# B&R Automation Studio project AutomatedPongGame (part 2)

#### basic.c
```c
/*******************************************************************
 * COPYRIGHT -- Bernecker + Rainer
 ********************************************************************
 * PROGRAM: Basic
 * File: Basic.c
 * Author: Bernecker + Rainer
 * Created: December 01, 2009
 ********************************************************************
 * Implementation of Program Basic
 ********************************************************************/

#ifdef _DEFAULT_INCLUDES
 #include <AsDefault.h>
#endif
#include <string.h>

/* defines of the state-constants */
#define STATE_WAIT              0
#define STATE_POWER_ON          1
#define STATE_HOME              2

#define STATE_READY             10
#define STATE_HALT              11
#define STATE_STOP              12
#define STATE_JOG_POSITIVE      13
#define STATE_JOG_NEGATIVE      14
#define STATE_MOVE_ABSOLUTE     15
#define STATE_MOVE_ADDITIVE     16
#define STATE_MOVE_VELOCITY     17

#define STATE_ERROR_AXIS        100
#define STATE_ERROR             101
#define STATE_ERROR_RESET       102

_INIT void BasicControl_init(void)
{

/* get axis object */
Axis1Obj = (UDINT)&gAxis01;

AxisStep = STATE_WAIT;  /* start step */

BasicControl.Parameter.Velocity              = 1000;  /*velocity for movement*/
BasicControl.Parameter.Acceleration          = 5000;  /*acceleration for movement*/
BasicControl.Parameter.Deceleration          = 5000;  /*deceleration for movement*/
BasicControl.Parameter.JogVelocity           = 400;   /*velocity for jogging */

}

_CYCLIC void BasicControl_cyclic(void)
{

/***************************************************************
        Control Sequence
***************************************************************/

/* status information is read before the step sequencer to attain a shorter reaction time */
/************************ MC_READSTATUS *************************/
MC_ReadStatus_0.Enable = !MC_ReadStatus_0.Error;
MC_ReadStatus_0.Axis = Axis1Obj;
MC_ReadStatus(&MC_ReadStatus_0);
BasicControl.AxisState.Disabled             = MC_ReadStatus_0.Disabled;
BasicControl.AxisState.StandStill           = MC_ReadStatus_0.StandStill;
BasicControl.AxisState.Stopping             = MC_ReadStatus_0.Stopping;
BasicControl.AxisState.Homing               = MC_ReadStatus_0.Homing;
BasicControl.AxisState.DiscreteMotion       = MC_ReadStatus_0.DiscreteMotion;
BasicControl.AxisState.ContinuousMotion     = MC_ReadStatus_0.ContinuousMotion;
BasicControl.AxisState.SynchronizedMotion   = MC_ReadStatus_0.SynchronizedMotion;
BasicControl.AxisState.ErrorStop            = MC_ReadStatus_0.Errorstop;

/********************MC_BR_READDRIVESTATUS***********************/
MC_BR_ReadDriveStatus_0.Enable = !MC_BR_ReadDriveStatus_0.Error;
MC_BR_ReadDriveStatus_0.Axis = Axis1Obj;
MC_BR_ReadDriveStatus_0.AdrDriveStatus = (UDINT)&(BasicControl.Status.DriveStatus);
MC_BR_ReadDriveStatus(&MC_BR_ReadDriveStatus_0);

/******************** MC_READACTUALPOSITION *********************/
MC_ReadActualPosition_0.Enable = (!MC_ReadActualPosition_0.Error);
MC_ReadActualPosition_0.Axis = Axis1Obj;
MC_ReadActualPosition(&MC_ReadActualPosition_0);
if(MC_ReadActualPosition_0.Valid == 1)
{
    BasicControl.Status.ActPosition = MC_ReadActualPosition_0.Position;
}

/******************** MC_READACTUALVELOCITY *********************/
MC_ReadActualVelocity_0.Enable = (!MC_ReadActualVelocity_0.Error);
MC_ReadActualVelocity_0.Axis = Axis1Obj;
MC_ReadActualVelocity(&MC_ReadActualVelocity_0);
if(MC_ReadActualVelocity_0.Valid == 1)
{
    BasicControl.Status.ActVelocity = MC_ReadActualVelocity_0.Velocity;
}

/************************ MC_READAXISERROR **********************/
MC_ReadAxisError_0.Enable = !MC_ReadAxisError_0.Error;
MC_ReadAxisError_0.Axis = Axis1Obj;
MC_ReadAxisError_0.DataAddress = (UDINT)&(BasicControl.Status.ErrorText);
MC_ReadAxisError_0.DataLength = sizeof(BasicControl.Status.ErrorText);
strcpy((void*)&MC_ReadAxisError_0.DataObjectName,"acp10etxen");
MC_ReadAxisError(&MC_ReadAxisError_0);

/**************** CHECK FOR GENERAL AXIS ERROR ******************/
    if ((MC_ReadAxisError_0.AxisErrorID != 0) && (MC_ReadAxisError_0.Valid == 1))
    {
        AxisStep = STATE_ERROR_AXIS;
    }
/***************** CHECK IF POWER SHOULD BE OFF *******************/
    else if ((BasicControl.Command.Power == 0) && (MC_ReadAxisError_0.Valid == 1))
    {
        if ((MC_ReadStatus_0.Errorstop == 1) && (MC_ReadStatus_0.Valid == 1))
        {
            AxisStep = STATE_ERROR_RESET;
        }
        else
        {
            AxisStep = STATE_WAIT;
        }
    }

/* central monitoring of stop command attains a shorter reaction time in case of emergency stop */
/******************CHECK for STOP COMMAND************************/
    if (BasicControl.Command.Stop == 1)
    {
        if ((AxisStep >= STATE_HOME) && (AxisStep <= STATE_ERROR))
        {
            /* reset all FB execute inputs we use */
            MC_Home_0.Execute = 0;
            MC_Stop_0.Execute = 0;
            MC_MoveAbsolute_0.Execute = 0;
            MC_MoveAdditive_0.Execute = 0;
            MC_MoveVelocity_0.Execute = 0;
            MC_Halt_0.Execute = 0;
            MC_ReadAxisError_0.Acknowledge = 0;
            MC_Reset_0.Execute = 0;

            /* reset user commands */
            BasicControl.Command.Halt = 0;
            BasicControl.Command.Home = 0;
            BasicControl.Command.MoveJogPos = 0;
            BasicControl.Command.MoveJogNeg = 0;
            BasicControl.Command.MoveVelocity = 0;
            BasicControl.Command.MoveAbsolute = 0;
            BasicControl.Command.MoveAdditive = 0;
            AxisStep = STATE_STOP;
        }
    }

switch(AxisStep)
{
/******************** WAIT *************************/
    case STATE_WAIT:  /* STATE: Wait */
        if (BasicControl.Command.Power == 1)
        {
            AxisStep = STATE_POWER_ON;
        }
        else
        {
            MC_Power_0.Enable = 0;
        }

        /* reset all FB execute inputs we use */
        MC_Home_0.Execute = 0;
        MC_Stop_0.Execute = 0;
        MC_MoveAbsolute_0.Execute = 0;
        MC_MoveAdditive_0.Execute = 0;
        MC_MoveVelocity_0.Execute = 0;
        MC_Halt_0.Execute = 0;
        MC_ReadAxisError_0.Acknowledge = 0;
        MC_Reset_0.Execute = 0;

        /* reset user commands */
        BasicControl.Command.Halt = 0;
        BasicControl.Command.Home = 0;
        BasicControl.Command.MoveJogPos = 0;
        BasicControl.Command.MoveJogNeg = 0;
        BasicControl.Command.MoveVelocity = 0;
        BasicControl.Command.MoveAbsolute = 0;
        BasicControl.Command.MoveAdditive = 0;

        BasicControl.Status.ErrorID = 0;
    break;

/******************** POWER ON **********************/
    case STATE_POWER_ON:  /* STATE: Power on */
        MC_Power_0.Enable = 1;
        if (MC_Power_0.Status == 1)
        {
            AxisStep = STATE_READY;
        }
        /* if a power error occured go to error state */
        if (MC_Power_0.Error == 1)
        {
            BasicControl.Status.ErrorID = MC_Power_0.ErrorID;
            AxisStep = STATE_ERROR;
        }
    break;

/******************** READY **********************/
    case STATE_READY:  /* STATE: Waiting for commands */
        if (BasicControl.Command.Home == 1)
        {
            BasicControl.Command.Home = 0;
            AxisStep = STATE_HOME;
        }
        else if (BasicControl.Command.Stop == 1)
        {
            AxisStep = STATE_STOP;
        }
        else if (BasicControl.Command.MoveJogPos == 1)
        {
            AxisStep = STATE_JOG_POSITIVE;
        }
        else if (BasicControl.Command.MoveJogNeg == 1)
        {
            AxisStep = STATE_JOG_NEGATIVE;
        }
        else if (BasicControl.Command.MoveAbsolute == 1)
        {
            BasicControl.Command.MoveAbsolute = 0;
            AxisStep = STATE_MOVE_ABSOLUTE;
        }
        else if (BasicControl.Command.MoveAdditive == 1)
        {
            BasicControl.Command.MoveAdditive = 0;
            AxisStep = STATE_MOVE_ADDITIVE;
        }
        else if (BasicControl.Command.MoveVelocity == 1)
        {
            BasicControl.Command.MoveVelocity = 0;
            AxisStep = STATE_MOVE_VELOCITY;
        }
        else if (BasicControl.Command.Halt == 1)
        {
            BasicControl.Command.Halt = 0;
            AxisStep = STATE_HALT;
        }
    break;

/******************** HOME **********************/
    case STATE_HOME:  /* STATE: start homing process */
        MC_Home_0.Position = BasicControl.Parameter.HomePosition;
        MC_Home_0.HomingMode = BasicControl.Parameter.HomeMode;
        MC_Home_0.Execute = 1;
        if (MC_Home_0.Done == 1)
        {
            MC_Home_0.Execute = 0;
            AxisStep = STATE_READY;
        }
        /* if a homing error occured go to error state */
        if (MC_Home_0.Error == 1)
        {
            MC_Home_0.Execute = 0;
            BasicControl.Status.ErrorID = MC_Home_0.ErrorID;
            AxisStep = STATE_ERROR;
        }
    break;

/************************HALT MOVEMENT**************************/
    case STATE_HALT:  /* STATE: Stop the active movement */
        MC_Halt_0.Deceleration = BasicControl.Parameter.Deceleration;
        MC_Halt_0.Execute = 1;
        if (MC_Halt_0.Done == 1)
        {
            MC_Halt_0.Execute = 0;
            AxisStep = STATE_READY;
        }
        /*check if error occured */
        if (MC_Halt_0.Error == 1)
        {
            MC_Halt_0.Execute = 0;
            BasicControl.Status.ErrorID = MC_Halt_0.ErrorID;
            AxisStep = STATE_ERROR;
        }
    break;

/*********************** STOP MOVEMENT *************************/
    case STATE_STOP: /* STATE: Stop movement as long as command is set */
        MC_Stop_0.Deceleration = BasicControl.Parameter.Deceleration;
        MC_Stop_0.Execute = 1;
        /* if axis is stopped go to ready state */
        if ((MC_Stop_0.Done == 1) && (BasicControl.Command.Stop == 0))
        {
            MC_Stop_0.Execute = 0;
            AxisStep = STATE_READY;
        }
        /* check if error occured */
        if (MC_Stop_0.Error == 1)
        {
            BasicControl.Status.ErrorID = MC_Stop_0.ErrorID;
            MC_Stop_0.Execute = 0;
            AxisStep = STATE_ERROR;
        }
    break;

/******************** START JOG MOVEMENT POSITVE **********************/
    case STATE_JOG_POSITIVE:  /* STATE: Start jog movement in positive direction */
        MC_MoveVelocity_0.Velocity      = BasicControl.Parameter.JogVelocity;
        MC_MoveVelocity_0.Acceleration  = BasicControl.Parameter.Acceleration;
        MC_MoveVelocity_0.Deceleration  = BasicControl.Parameter.Deceleration;
        MC_MoveVelocity_0.Direction     = mcPOSITIVE_DIR;
        MC_MoveVelocity_0.Execute = 1;
        /* check if jog movement should be stopped */
        if (BasicControl.Command.MoveJogPos == 0)
        {
            MC_MoveVelocity_0.Execute = 0;
            AxisStep = STATE_HALT;
        }
        /* check if error occured */
        if (MC_MoveVelocity_0.Error == 1)
        {
            BasicControl.Status.ErrorID = MC_MoveVelocity_0.ErrorID;
            MC_MoveVelocity_0.Execute = 0;
            AxisStep = STATE_ERROR;
        }
    break;

/******************** START JOG MOVEMENT NEGATIVE **********************/
    case STATE_JOG_NEGATIVE:  /* STATE: Start jog movement in negative direction */
        MC_MoveVelocity_0.Velocity      = BasicControl.Parameter.JogVelocity;
        MC_MoveVelocity_0.Acceleration  = BasicControl.Parameter.Acceleration;
        MC_MoveVelocity_0.Deceleration  = BasicControl.Parameter.Deceleration;
        MC_MoveVelocity_0.Direction     = mcNEGATIVE_DIR;
        MC_MoveVelocity_0.Execute = 1;
        /* check if jog movement should be stopped */
        if (BasicControl.Command.MoveJogNeg == 0)
        {
            MC_MoveVelocity_0.Execute = 0;
            AxisStep = STATE_HALT;
        }
        /* check if error occured */
        if (MC_MoveVelocity_0.Error == 1)
        {
            BasicControl.Status.ErrorID = MC_MoveVelocity_0.ErrorID;
            MC_MoveVelocity_0.Execute = 0;
            AxisStep = STATE_ERROR;
        }
    break;

/******************** START ABSOLUTE MOVEMENT **********************/
    case STATE_MOVE_ABSOLUTE:  /* STATE: Start absolute movement */
        MC_MoveAbsolute_0.Position      = BasicControl.Parameter.Position;
        MC_MoveAbsolute_0.Velocity      = BasicControl.Parameter.Velocity;
        MC_MoveAbsolute_0.Acceleration  = BasicControl.Parameter.Acceleration;
        MC_MoveAbsolute_0.Deceleration  = BasicControl.Parameter.Deceleration;
        MC_MoveAbsolute_0.Direction     = BasicControl.Parameter.Direction;
        MC_MoveAbsolute_0.Execute = 1;
        /* check if commanded position is reached */
        if (BasicControl.Command.Halt == 1)
        {
            BasicControl.Command.Halt = 0;
            MC_MoveAbsolute_0.Execute = 0;
            AxisStep = STATE_HALT;
        }
        else if (MC_MoveAbsolute_0.Done == 1)
        {
            MC_MoveAbsolute_0.Execute = 0;
             AxisStep = STATE_READY;
        }
        /* check if error occured */
        if (MC_MoveAbsolute_0.Error == 1)
        {
            BasicControl.Status.ErrorID = MC_MoveAbsolute_0.ErrorID;
            MC_MoveAbsolute_0.Execute = 0;
            AxisStep = STATE_ERROR;
        }
    break;

/******************** START ADDITIVE MOVEMENT **********************/
    case STATE_MOVE_ADDITIVE:  /* STATE: Start additive movement */
        MC_MoveAdditive_0.Distance      = BasicControl.Parameter.Distance;
        MC_MoveAdditive_0.Velocity      = BasicControl.Parameter.Velocity;
        MC_MoveAdditive_0.Acceleration  = BasicControl.Parameter.Acceleration;
        MC_MoveAdditive_0.Deceleration  = BasicControl.Parameter.Deceleration;
        MC_MoveAdditive_0.Execute = 1;
        /* check if commanded distance is reached */
        if (BasicControl.Command.Halt == 1)
        {
            BasicControl.Command.Halt = 0;
            MC_MoveAdditive_0.Execute = 0;
            AxisStep = STATE_HALT;
        }
        else if (MC_MoveAdditive_0.Done == 1)
        {
            MC_MoveAdditive_0.Execute = 0;
             AxisStep = STATE_READY;
        }
        /* check if error occured */
        if (MC_MoveAdditive_0.Error == 1)
        {
            BasicControl.Status.ErrorID = MC_MoveAdditive_0.ErrorID;
            MC_MoveAdditive_0.Execute = 0;
            AxisStep = STATE_ERROR;
        }
    break;

/******************** START VELOCITY MOVEMENT **********************/
    case STATE_MOVE_VELOCITY:  /* STATE: Start velocity movement */
        MC_MoveVelocity_0.Velocity      = BasicControl.Parameter.Velocity;
        MC_MoveVelocity_0.Acceleration  = BasicControl.Parameter.Acceleration;
        MC_MoveVelocity_0.Deceleration  = BasicControl.Parameter.Deceleration;
        MC_MoveVelocity_0.Direction     = BasicControl.Parameter.Direction;
        MC_MoveVelocity_0.Execute = 1;
        /* check if commanded velocity is reached */
        if (BasicControl.Command.Halt == 1)
        {
            BasicControl.Command.Halt = 0;
            MC_MoveVelocity_0.Execute = 0;
            AxisStep = STATE_HALT;
        }
        else if (MC_MoveVelocity_0.InVelocity == 1)
        {
            MC_MoveVelocity_0.Execute = 0;
             AxisStep = STATE_READY;
        }
        /* check if error occured */
        if (MC_MoveVelocity_0.Error == 1)
        {
            BasicControl.Status.ErrorID = MC_MoveVelocity_0.ErrorID;
            MC_MoveVelocity_0.Execute = 0;
            AxisStep = STATE_ERROR;
        }
    break;

/******************** FB-ERROR OCCURED *************************/
    case STATE_ERROR:  /* STATE: Error */
        /* check if FB indicates an axis error */
        if (MC_ReadAxisError_0.AxisErrorCount != 0)
        {
            AxisStep = STATE_ERROR_AXIS;
        }
        else
        {
            if (BasicControl.Command.ErrorAcknowledge == 1)
            {
                BasicControl.Command.ErrorAcknowledge = 0;
                BasicControl.Status.ErrorID = 0;
                /* reset axis if it is in axis state ErrorStop */
                if ((MC_ReadStatus_0.Errorstop == 1) && (MC_ReadStatus_0.Valid == 1))
                {
                    AxisStep = STATE_ERROR_RESET;
                }
                else
                {
                    AxisStep = STATE_WAIT;
                }
            }
        }
    break;

/******************** AXIS-ERROR OCCURED *************************/
    case STATE_ERROR_AXIS:  /* STATE: Axis Error */
        if (MC_ReadAxisError_0.Valid == 1)
        {
            if (MC_ReadAxisError_0.AxisErrorID != 0)
            {
                BasicControl.Status.ErrorID = MC_ReadAxisError_0.AxisErrorID;
            }
            MC_ReadAxisError_0.Acknowledge = 0;
            if (BasicControl.Command.ErrorAcknowledge == 1)
            {
                BasicControl.Command.ErrorAcknowledge = 0;
                /* acknowledge axis error */
                if (MC_ReadAxisError_0.AxisErrorID != 0)
                {
                    MC_ReadAxisError_0.Acknowledge = 1;
                }
            }
            if (MC_ReadAxisError_0.AxisErrorCount == 0)
            {
                BasicControl.Status.ErrorID = 0;
                /* reset axis if it is in axis state ErrorStop */
                if ((MC_ReadStatus_0.Errorstop == 1) && (MC_ReadStatus_0.Valid == 1))
                {
                    AxisStep = STATE_ERROR_RESET;
                }
                else
                {
                    AxisStep = STATE_WAIT;
                }
            }
        }
    break;

/******************** RESET DONE *************************/
    case STATE_ERROR_RESET:  /* STATE: Wait for reset done */
        MC_Reset_0.Execute = 1;
        /* reset MC_Power.Enable if this FB is in Error*/
        if(MC_Power_0.Error == 1)
        {
            MC_Power_0.Enable = 0;
        }
        if(MC_Reset_0.Done == 1)
        {
            MC_Reset_0.Execute = 0;
            AxisStep = STATE_WAIT;
        }
        else if (MC_Reset_0.Error == 1)
        {
            MC_Reset_0.Execute = 0;
            AxisStep = STATE_ERROR;
        }
    break;

/******************** SEQUENCE END *************************/
}

/***************************************************************
        Function Block Calls
***************************************************************/

/************************** MC_POWER ****************************/
MC_Power_0.Axis = Axis1Obj;  /* pointer to axis */
MC_Power(&MC_Power_0);

/************************** MC_HOME *****************************/
MC_Home_0.Axis = Axis1Obj;
MC_Home(&MC_Home_0);

/********************** MC_MOVEABSOLUTE *************************/
MC_MoveAbsolute_0.Axis = Axis1Obj;
MC_MoveAbsolute(&MC_MoveAbsolute_0);

/********************** MC_MOVEADDITIVE *************************/
MC_MoveAdditive_0.Axis = Axis1Obj;
MC_MoveAdditive(&MC_MoveAdditive_0);

/********************** MC_MOVEVELOCITY *************************/
MC_MoveVelocity_0.Axis = Axis1Obj;
MC_MoveVelocity(&MC_MoveVelocity_0);

/************************** MC_STOP *****************************/
MC_Stop_0.Axis = Axis1Obj;
MC_Stop(&MC_Stop_0);

/**************************MC_HALT*******************************/
MC_Halt_0.Axis = Axis1Obj;
MC_Halt(&MC_Halt_0);

/************************** MC_RESET ****************************/
MC_Reset_0.Axis = Axis1Obj;
MC_Reset(&MC_Reset_0);

}
```

#### Cyclic.cpp
```cpp
#ifdef _DEFAULT_INCLUDES
	#include <AsDefault.h>
#endif
#include <string.h>

/* defines of the state-constants */
#define STATE_WAIT              0
#define STATE_POWER_ON          1
#define STATE_HOME              2

#define STATE_READY             10
#define STATE_HALT              11
#define STATE_STOP              12
#define STATE_JOG_POSITIVE      13
#define STATE_JOG_NEGATIVE      14
#define STATE_MOVE_ABSOLUTE     15
#define STATE_MOVE_ADDITIVE     16
#define STATE_MOVE_VELOCITY     17

#define STATE_ERROR_AXIS        100
#define STATE_ERROR             101
#define STATE_ERROR_RESET       102

#define RED_COLOR 51
#define GREEN_COLOR 10

#define MIDDELPUNT_TRAPPER_OFFSET 15
//#define ACTPOSITION_TO_MM 0.0784

unsigned long bur_heap_size = 0xFFFF;

void _CYCLIC ProgramCyclic(void)
{
	/***************************************************************
        Control Sequence
	***************************************************************/

	/* status information is read before the step sequencer to attain a shorter reaction time */
	/************************ MC_READSTATUS *************************/
	MC_ReadStatus_0.Enable = !MC_ReadStatus_0.Error;
	MC_ReadStatus_0.Axis = Axis1Obj;
	MC_ReadStatus(&MC_ReadStatus_0);
	BasicControl.AxisState.Disabled             = MC_ReadStatus_0.Disabled;
	BasicControl.AxisState.StandStill           = MC_ReadStatus_0.StandStill;
	BasicControl.AxisState.Stopping             = MC_ReadStatus_0.Stopping;
	BasicControl.AxisState.Homing               = MC_ReadStatus_0.Homing;
	BasicControl.AxisState.DiscreteMotion       = MC_ReadStatus_0.DiscreteMotion;
	BasicControl.AxisState.ContinuousMotion     = MC_ReadStatus_0.ContinuousMotion;
	BasicControl.AxisState.SynchronizedMotion   = MC_ReadStatus_0.SynchronizedMotion;
	BasicControl.AxisState.ErrorStop            = MC_ReadStatus_0.Errorstop;

	/********************MC_BR_READDRIVESTATUS***********************/
	MC_BR_ReadDriveStatus_0.Enable = !MC_BR_ReadDriveStatus_0.Error;
	MC_BR_ReadDriveStatus_0.Axis = Axis1Obj;
	MC_BR_ReadDriveStatus_0.AdrDriveStatus = (UDINT)&(BasicControl.Status.DriveStatus);
	MC_BR_ReadDriveStatus(&MC_BR_ReadDriveStatus_0);

	/******************** MC_READACTUALPOSITION *********************/
	MC_ReadActualPosition_0.Enable = (!MC_ReadActualPosition_0.Error);
	MC_ReadActualPosition_0.Axis = Axis1Obj;
	MC_ReadActualPosition(&MC_ReadActualPosition_0);
	if(MC_ReadActualPosition_0.Valid == 1)
	{
		BasicControl.Status.ActPosition = MC_ReadActualPosition_0.Position;
	}

	/******************** MC_READACTUALVELOCITY *********************/
	MC_ReadActualVelocity_0.Enable = (!MC_ReadActualVelocity_0.Error);
	MC_ReadActualVelocity_0.Axis = Axis1Obj;
	MC_ReadActualVelocity(&MC_ReadActualVelocity_0);
	if(MC_ReadActualVelocity_0.Valid == 1)
	{
		BasicControl.Status.ActVelocity = MC_ReadActualVelocity_0.Velocity;
	}

	/************************ MC_READAXISERROR **********************/
	MC_ReadAxisError_0.Enable = !MC_ReadAxisError_0.Error;
	MC_ReadAxisError_0.Axis = Axis1Obj;
	MC_ReadAxisError_0.DataAddress = (UDINT)&(BasicControl.Status.ErrorText);
	MC_ReadAxisError_0.DataLength = sizeof(BasicControl.Status.ErrorText);
	strcpy(MC_ReadAxisError_0.DataObjectName,"acp10etxen");
	MC_ReadAxisError(&MC_ReadAxisError_0);

	/**************** CHECK FOR GENERAL AXIS ERROR ******************/
	if ((MC_ReadAxisError_0.AxisErrorID != 0) && (MC_ReadAxisError_0.Valid == 1))
	{
		AxisStep = STATE_ERROR_AXIS;
	}
		/***************** CHECK IF POWER SHOULD BE OFF *******************/
	else if ((BasicControl.Command.Power == 0) && (MC_ReadAxisError_0.Valid == 1))
	{
		if ((MC_ReadStatus_0.Errorstop == 1) && (MC_ReadStatus_0.Valid == 1))
		{
			AxisStep = STATE_ERROR_RESET;
		}
		else
		{
			AxisStep = STATE_WAIT;
		}
	}

	/* central monitoring of stop command attains a shorter reaction time in case of emergency stop */
	/******************CHECK for STOP COMMAND************************/
	if (BasicControl.Command.Stop == 1)
	{
		if ((AxisStep >= STATE_HOME) && (AxisStep <= STATE_ERROR))
		{
			/* reset all FB execute inputs we use */
			MC_Home_0.Execute = 0;
			MC_Stop_0.Execute = 0;
			MC_MoveAbsolute_0.Execute = 0;
			MC_MoveAdditive_0.Execute = 0;
			MC_MoveVelocity_0.Execute = 0;
			MC_Halt_0.Execute = 0;
			MC_ReadAxisError_0.Acknowledge = 0;
			MC_Reset_0.Execute = 0;

			/* reset user commands */
			BasicControl.Command.Halt = 0;
			BasicControl.Command.Home = 0;
			BasicControl.Command.MoveJogPos = 0;
			BasicControl.Command.MoveJogNeg = 0;
			BasicControl.Command.MoveVelocity = 0;
			BasicControl.Command.MoveAbsolute = 0;
			BasicControl.Command.MoveAdditive = 0;
			AxisStep = STATE_STOP;
		}
	}

	switch(AxisStep)
	{
		/******************** WAIT *************************/
		case STATE_WAIT:  /* STATE: Wait */
			if (BasicControl.Command.Power == 1)
			{
				AxisStep = STATE_POWER_ON;
			}
			else
			{
				MC_Power_0.Enable = 0;
			}

			/* reset all FB execute inputs we use */
			MC_Home_0.Execute = 0;
			MC_Stop_0.Execute = 0;
			MC_MoveAbsolute_0.Execute = 0;
			MC_MoveAdditive_0.Execute = 0;
			MC_MoveVelocity_0.Execute = 0;
			MC_Halt_0.Execute = 0;
			MC_ReadAxisError_0.Acknowledge = 0;
			MC_Reset_0.Execute = 0;

			/* reset user commands */
			BasicControl.Command.Halt = 0;
			BasicControl.Command.Home = 0;
			BasicControl.Command.MoveJogPos = 0;
			BasicControl.Command.MoveJogNeg = 0;
			BasicControl.Command.MoveVelocity = 0;
			BasicControl.Command.MoveAbsolute = 0;
			BasicControl.Command.MoveAdditive = 0;

			BasicControl.Status.ErrorID = 0;
			break;

		/******************** POWER ON **********************/
		case STATE_POWER_ON:  /* STATE: Power on */
			MC_Power_0.Enable = 1;
			if (MC_Power_0.Status == 1)
			{
				AxisStep = STATE_READY;
			}
			/* if a power error occured go to error state */
			if (MC_Power_0.Error == 1)
			{
				BasicControl.Status.ErrorID = MC_Power_0.ErrorID;
				AxisStep = STATE_ERROR;
			}
			break;

		/******************** READY **********************/
		case STATE_READY:  /* STATE: Waiting for commands */
			if (BasicControl.Command.Home == 1)
			{
				BasicControl.Command.Home = 0;
				AxisStep = STATE_HOME;
			}
			else if (BasicControl.Command.Stop == 1)
			{
				AxisStep = STATE_STOP;
			}
			else if (BasicControl.Command.MoveJogPos == 1)
			{
				AxisStep = STATE_JOG_POSITIVE;
			}
			else if (BasicControl.Command.MoveJogNeg == 1)
			{
				AxisStep = STATE_JOG_NEGATIVE;
			}
			else if (BasicControl.Command.MoveAbsolute == 1)
			{
				BasicControl.Command.MoveAbsolute = 0;
				AxisStep = STATE_MOVE_ABSOLUTE;
			}
			else if (BasicControl.Command.MoveAdditive == 1)
			{
				BasicControl.Command.MoveAdditive = 0;
				AxisStep = STATE_MOVE_ADDITIVE;
			}
			else if (BasicControl.Command.MoveVelocity == 1)
			{
				BasicControl.Command.MoveVelocity = 0;
				AxisStep = STATE_MOVE_VELOCITY;
			}
			else if (BasicControl.Command.Halt == 1)
			{
				BasicControl.Command.Halt = 0;
				AxisStep = STATE_HALT;
			}
			break;

		/******************** HOME **********************/
		case STATE_HOME:  /* STATE: start homing process */
			MC_Home_0.Position = BasicControl.Parameter.HomePosition;
			MC_Home_0.HomingMode = BasicControl.Parameter.HomeMode;
			MC_Home_0.Execute = 1;
			if (MC_Home_0.Done == 1)
			{
				MC_Home_0.Execute = 0;
				AxisStep = STATE_READY;
			}
			/* if a homing error occured go to error state */
			if (MC_Home_0.Error == 1)
			{
				MC_Home_0.Execute = 0;
				BasicControl.Status.ErrorID = MC_Home_0.ErrorID;
				AxisStep = STATE_ERROR;
			}
			break;

		/************************HALT MOVEMENT**************************/
		case STATE_HALT:  /* STATE: Stop the active movement */
			MC_Halt_0.Deceleration = BasicControl.Parameter.Deceleration;
			MC_Halt_0.Execute = 1;
			if (MC_Halt_0.Done == 1)
			{
				MC_Halt_0.Execute = 0;
				AxisStep = STATE_READY;
			}
			/*check if error occured */
			if (MC_Halt_0.Error == 1)
			{
				MC_Halt_0.Execute = 0;
				BasicControl.Status.ErrorID = MC_Halt_0.ErrorID;
				AxisStep = STATE_ERROR;
			}
			break;

		/*********************** STOP MOVEMENT *************************/
		case STATE_STOP: /* STATE: Stop movement as long as command is set */
			MC_Stop_0.Deceleration = BasicControl.Parameter.Deceleration;
			MC_Stop_0.Execute = 1;
			/* if axis is stopped go to ready state */
			if ((MC_Stop_0.Done == 1) && (BasicControl.Command.Stop == 0))
			{
				MC_Stop_0.Execute = 0;
				AxisStep = STATE_READY;
			}
			/* check if error occured */
			if (MC_Stop_0.Error == 1)
			{
				BasicControl.Status.ErrorID = MC_Stop_0.ErrorID;
				MC_Stop_0.Execute = 0;
				AxisStep = STATE_ERROR;
			}
			break;

		/******************** START JOG MOVEMENT POSITVE **********************/
		case STATE_JOG_POSITIVE:  /* STATE: Start jog movement in positive direction */
			MC_MoveVelocity_0.Velocity      = BasicControl.Parameter.JogVelocity;
			MC_MoveVelocity_0.Acceleration  = BasicControl.Parameter.Acceleration;
			MC_MoveVelocity_0.Deceleration  = BasicControl.Parameter.Deceleration;
			MC_MoveVelocity_0.Direction     = mcPOSITIVE_DIR;
			MC_MoveVelocity_0.Execute = 1;
			/* check if jog movement should be stopped */
			if (BasicControl.Command.MoveJogPos == 0)
			{
				MC_MoveVelocity_0.Execute = 0;
				AxisStep = STATE_HALT;
			}
			/* check if error occured */
			if (MC_MoveVelocity_0.Error == 1)
			{
				BasicControl.Status.ErrorID = MC_MoveVelocity_0.ErrorID;
				MC_MoveVelocity_0.Execute = 0;
				AxisStep = STATE_ERROR;
			}
			break;

		/******************** START JOG MOVEMENT NEGATIVE **********************/
		case STATE_JOG_NEGATIVE:  /* STATE: Start jog movement in negative direction */
			MC_MoveVelocity_0.Velocity      = BasicControl.Parameter.JogVelocity;
			MC_MoveVelocity_0.Acceleration  = BasicControl.Parameter.Acceleration;
			MC_MoveVelocity_0.Deceleration  = BasicControl.Parameter.Deceleration;
			MC_MoveVelocity_0.Direction     = mcNEGATIVE_DIR;
			MC_MoveVelocity_0.Execute = 1;
			/* check if jog movement should be stopped */
			if (BasicControl.Command.MoveJogNeg == 0)
			{
				MC_MoveVelocity_0.Execute = 0;
				AxisStep = STATE_HALT;
			}
			/* check if error occured */
			if (MC_MoveVelocity_0.Error == 1)
			{
				BasicControl.Status.ErrorID = MC_MoveVelocity_0.ErrorID;
				MC_MoveVelocity_0.Execute = 0;
				AxisStep = STATE_ERROR;
			}
			break;

		/******************** START ABSOLUTE MOVEMENT **********************/
		case STATE_MOVE_ABSOLUTE:  /* STATE: Start absolute movement */
			MC_MoveAbsolute_0.Position      = BasicControl.Parameter.Position;
			MC_MoveAbsolute_0.Velocity      = BasicControl.Parameter.Velocity;
			MC_MoveAbsolute_0.Acceleration  = BasicControl.Parameter.Acceleration;
			MC_MoveAbsolute_0.Deceleration  = BasicControl.Parameter.Deceleration;
			MC_MoveAbsolute_0.Direction     = BasicControl.Parameter.Direction;
			MC_MoveAbsolute_0.Execute = 1;
			/* check if commanded position is reached */
			if (BasicControl.Command.Halt == 1)
			{
				BasicControl.Command.Halt = 0;
				MC_MoveAbsolute_0.Execute = 0;
				AxisStep = STATE_HALT;
			}
			else if (MC_MoveAbsolute_0.Done == 1)
			{
				MC_MoveAbsolute_0.Execute = 0;
				AxisStep = STATE_READY;
			}
			/* check if error occured */
			if (MC_MoveAbsolute_0.Error == 1)
			{
				BasicControl.Status.ErrorID = MC_MoveAbsolute_0.ErrorID;
				MC_MoveAbsolute_0.Execute = 0;
				AxisStep = STATE_ERROR;
			}
			break;

		/******************** START ADDITIVE MOVEMENT **********************/
		case STATE_MOVE_ADDITIVE:  /* STATE: Start additive movement */
			MC_MoveAdditive_0.Distance      = BasicControl.Parameter.Distance;
			MC_MoveAdditive_0.Velocity      = BasicControl.Parameter.Velocity;
			MC_MoveAdditive_0.Acceleration  = BasicControl.Parameter.Acceleration;
			MC_MoveAdditive_0.Deceleration  = BasicControl.Parameter.Deceleration;
			MC_MoveAdditive_0.Execute = 1;
			/* check if commanded distance is reached */
			if (BasicControl.Command.Halt == 1)
			{
				BasicControl.Command.Halt = 0;
				MC_MoveAdditive_0.Execute = 0;
				AxisStep = STATE_HALT;
			}
			else if (MC_MoveAdditive_0.Done == 1)
			{
				MC_MoveAdditive_0.Execute = 0;
				AxisStep = STATE_READY;
			}
			/* check if error occured */
			if (MC_MoveAdditive_0.Error == 1)
			{
				BasicControl.Status.ErrorID = MC_MoveAdditive_0.ErrorID;
				MC_MoveAdditive_0.Execute = 0;
				AxisStep = STATE_ERROR;
			}
			break;

		/******************** START VELOCITY MOVEMENT **********************/
		case STATE_MOVE_VELOCITY:  /* STATE: Start velocity movement */
			MC_MoveVelocity_0.Velocity      = BasicControl.Parameter.Velocity;
			MC_MoveVelocity_0.Acceleration  = BasicControl.Parameter.Acceleration;
			MC_MoveVelocity_0.Deceleration  = BasicControl.Parameter.Deceleration;
			MC_MoveVelocity_0.Direction     = BasicControl.Parameter.Direction;
			MC_MoveVelocity_0.Execute = 1;
			/* check if commanded velocity is reached */
			if (BasicControl.Command.Halt == 1)
			{
				BasicControl.Command.Halt = 0;
				MC_MoveVelocity_0.Execute = 0;
				AxisStep = STATE_HALT;
			}
			else if (MC_MoveVelocity_0.InVelocity == 1)
			{
				MC_MoveVelocity_0.Execute = 0;
				AxisStep = STATE_READY;
			}
			/* check if error occured */
			if (MC_MoveVelocity_0.Error == 1)
			{
				BasicControl.Status.ErrorID = MC_MoveVelocity_0.ErrorID;
				MC_MoveVelocity_0.Execute = 0;
				AxisStep = STATE_ERROR;
			}
			break;

		/******************** FB-ERROR OCCURED *************************/
		case STATE_ERROR:  /* STATE: Error */
			/* check if FB indicates an axis error */
			if (MC_ReadAxisError_0.AxisErrorCount != 0)
			{
				AxisStep = STATE_ERROR_AXIS;
			}
			else
			{
				if (BasicControl.Command.ErrorAcknowledge == 1)
				{
					BasicControl.Command.ErrorAcknowledge = 0;
					BasicControl.Status.ErrorID = 0;
					/* reset axis if it is in axis state ErrorStop */
					if ((MC_ReadStatus_0.Errorstop == 1) && (MC_ReadStatus_0.Valid == 1))
					{
						AxisStep = STATE_ERROR_RESET;
					}
					else
					{
						AxisStep = STATE_WAIT;
					}
				}
			}
			break;

		/******************** AXIS-ERROR OCCURED *************************/
		case STATE_ERROR_AXIS:  /* STATE: Axis Error */
			if (MC_ReadAxisError_0.Valid == 1)
			{
				if (MC_ReadAxisError_0.AxisErrorID != 0)
				{
					BasicControl.Status.ErrorID = MC_ReadAxisError_0.AxisErrorID;
				}
				MC_ReadAxisError_0.Acknowledge = 0;
				if (BasicControl.Command.ErrorAcknowledge == 1)
				{
					BasicControl.Command.ErrorAcknowledge = 0;
					/* acknowledge axis error */
					if (MC_ReadAxisError_0.AxisErrorID != 0)
					{
						MC_ReadAxisError_0.Acknowledge = 1;
					}
				}
				if (MC_ReadAxisError_0.AxisErrorCount == 0)
				{
					BasicControl.Status.ErrorID = 0;
					/* reset axis if it is in axis state ErrorStop */
					if ((MC_ReadStatus_0.Errorstop == 1) && (MC_ReadStatus_0.Valid == 1))
					{
						AxisStep = STATE_ERROR_RESET;
					}
					else
					{
						AxisStep = STATE_WAIT;
					}
				}
			}
			break;

		/******************** RESET DONE *************************/
		case STATE_ERROR_RESET:  /* STATE: Wait for reset done */
			MC_Reset_0.Execute = 1;
			/* reset MC_Power.Enable if this FB is in Error*/
			if(MC_Power_0.Error == 1)
			{
				MC_Power_0.Enable = 0;
			}
			if(MC_Reset_0.Done == 1)
			{
				MC_Reset_0.Execute = 0;
				AxisStep = STATE_WAIT;
			}
			else if (MC_Reset_0.Error == 1)
			{
				MC_Reset_0.Execute = 0;
				AxisStep = STATE_ERROR;
			}
			break;

		/******************** SEQUENCE END *************************/
	}

/***************************************************************
        Function Block Calls
***************************************************************/

/************************** MC_POWER ****************************/
	MC_Power_0.Axis = Axis1Obj;  /* pointer to axis */
	MC_Power(&MC_Power_0);

	/************************** MC_HOME *****************************/
	MC_Home_0.Axis = Axis1Obj;
	MC_Home(&MC_Home_0);

	/********************** MC_MOVEABSOLUTE *************************/
	MC_MoveAbsolute_0.Axis = Axis1Obj;
	MC_MoveAbsolute(&MC_MoveAbsolute_0);

	/********************** MC_MOVEADDITIVE *************************/
	MC_MoveAdditive_0.Axis = Axis1Obj;
	MC_MoveAdditive(&MC_MoveAdditive_0);

	/********************** MC_MOVEVELOCITY *************************/
	MC_MoveVelocity_0.Axis = Axis1Obj;
	MC_MoveVelocity(&MC_MoveVelocity_0);

	/************************** MC_STOP *****************************/
	MC_Stop_0.Axis = Axis1Obj;
	MC_Stop(&MC_Stop_0);

	/**************************MC_HALT*******************************/
	MC_Halt_0.Axis = Axis1Obj;
	MC_Halt(&MC_Halt_0);

	/************************** MC_RESET ****************************/
	MC_Reset_0.Axis = Axis1Obj;
	MC_Reset(&MC_Reset_0);

	hmiActPosition = ActPositionToMM(BasicControl.Status.ActPosition); //function

	digitalOutputs = SetOutputs(digitalOutputs, turnOnVentilator, turnOnSolenoid); //function

	if(incrementTrapperSpeed && BasicControl.Parameter.JogVelocity < 4000)
	{
		BasicControl.Parameter.JogVelocity++;
	}
	if(decrementTrapperSpeed && BasicControl.Parameter.JogVelocity > 0)
	{
		BasicControl.Parameter.JogVelocity--;
	}

	if(incrementTrapperAccDecc && BasicControl.Parameter.Acceleration < 50000)
	{
		BasicControl.Parameter.Acceleration += 10;
		BasicControl.Parameter.Deceleration += 10;
	}
	if(decrementTrapperAccDecc && BasicControl.Parameter.Acceleration > 100)
	{
		BasicControl.Parameter.Acceleration -= 10;
		BasicControl.Parameter.Deceleration -= 10;
	}
}
```

#### Init.cpp
```cpp
#ifdef _DEFAULT_INCLUDES
	#include <AsDefault.h>
#endif
#include <string.h>

#define STATE_WAIT              0

void _INIT ProgramInit(void)
{
	/* get axis object */
	Axis1Obj = (UDINT)&gAxis01;

	AxisStep = STATE_WAIT;  /* start step */

	BasicControl.Parameter.Velocity              = 1000;  /*velocity for movement*/
	BasicControl.Parameter.Acceleration          = 5000;  /*acceleration for movement*/
	BasicControl.Parameter.Deceleration          = 5000;  /*deceleration for movement*/
	BasicControl.Parameter.JogVelocity           = 400;   /*velocity for jogging */

}
```

### Data object Logical/gAxis01obj/gAxis01i (Ax)

#### gAxis01i.ax
```
InitParameter (Version=5.30.2, NcSwId=ACP10)
  ACP10AXIS_typ:
    dig_in:
      level:
        reference = ncACTIV_HI
        pos_hw_end = ncACTIV_HI
        neg_hw_end = ncACTIV_HI
        trigger1 = ncACTIV_HI
        trigger2 = ncACTIV_HI
    encoder_if:
      parameter:
        count_dir = ncSTANDARD
        scaling:
          load:
            units = 1000
            rev_motor = 1
    limit:
      parameter:
        v_pos = 10000.0
        v_neg = 10000.0
        a1_pos = 50000.0
        a2_pos = 50000.0
        a1_neg = 50000.0
        a2_neg = 50000.0
        t_jolt = 0.0
        t_in_pos = 0.0
        pos_sw_end = 8388607
        neg_sw_end = -8388608
        ds_warning = 500.0
        ds_stop = 1000.0
        a_stop = 1.0E+30
        dv_stop = 0.0
        dv_stop_mode = ncOFF
    controller:
      mode = ncPOSITION
      position:
        kv = 123.0
        tn = 0.0
        t_predict = 0.0004
        t_total = 0.0004
        p_max = 1.0E+30
        i_max = 0.0
      speed:
        kv = 0.15
        tn = 0.0
        t_filter = 0.0
        isq_filter1:
          type = ncOFF
          a0 = 0.0
          a1 = 0.0
          b0 = 0.0
          b1 = 0.0
          b2 = 0.0
          c0_par_id = 0
          c1_par_id = 0
        isq_filter2:
          type = ncOFF
          a0 = 0.0
          a1 = 0.0
          b0 = 0.0
          b1 = 0.0
          b2 = 0.0
          c0_par_id = 0
          c1_par_id = 0
        isq_filter3:
          type = ncOFF
          a0 = 0.0
          a1 = 0.0
          b0 = 0.0
          b1 = 0.0
          b2 = 0.0
          c0_par_id = 0
          c1_par_id = 0
      uf:
        type = ncLINEAR + ncCORRECTION
        auto_config = ncMOTOR_PAR
        u0 = 0.0
        un = 0.0
        fn = 50.0
        k_f_slip = 0.0
      ff:
        mode = ncSTANDARD
        torque_load = 0.0
        torque_pos = 0.0
        torque_neg = 0.0
        kv_torque = 0.0
        inertia = 0.0
        t_filter_a = 0.0
      fb:
        mode = ncSTANDARD
        speed_mix_ratio = 0.0
        speed_kv = 0.0
      model:
        mass1:
          inertia = 0.0
          viscous_friction = 0.0
        mass2:
          inertia = 0.0
          viscous_friction = 0.0
          stiffness = 0.0
          damping = 0.0
    move:
      stop:
        parameter[0]:
          decel_ramp = ncA_LIMIT
          controller = ncON
        parameter[1]:
          decel_ramp = ncA_LIMIT
          controller = ncON
        parameter[2]:
          decel_ramp = ncA_LIMIT
          controller = ncON
        parameter[3]:
          decel_ramp = ncA_LIMIT
          controller = ncON
        quickstop:
          decel_ramp = ncA_LIMIT
          t_jolt = 0.0
        drive_error:
          decel_ramp = ncA_LIMIT
      homing:
        parameter:
          s = 1000
          v_switch = 5000.0
          v_trigger = 500.0
          a = 50000.0
          mode = ncDIRECT
          edge_sw = ncPOSITIVE
          start_dir = ncPOSITIVE
          trigg_dir = ncPOSITIVE
          ref_pulse = ncOFF
          fix_dir = ncOFF
          tr_s_block = 0.0
          torque_lim = 0.0
          ds_block = 0.0
          ds_stop = 0.0
      basis:
        parameter:
          v_pos = 5000.0
          v_neg = 5000.0
          a1_pos = 50000.0
          a2_pos = 50000.0
          a1_neg = 50000.0
          a2_neg = 50000.0
    message:
      text:
        parameter:
          format = ncBREAK
          columns = 80
          data_modul = acp10etxen
```

### Package Logical/gAxis02obj - gAxis02obj

### Data object Logical/gAxis02obj/gAxis02i (Ax)

#### gAxis02i.ax
```
InitParameter (Version=5.30.2, NcSwId=ACP10)
  ACP10AXIS_typ:
    dig_in:
      level:
        reference = ncACTIV_HI
        pos_hw_end = ncACTIV_HI
        neg_hw_end = ncACTIV_HI
        trigger1 = ncACTIV_HI
        trigger2 = ncACTIV_HI
    encoder_if:
      parameter:
        count_dir = ncSTANDARD
        scaling:
          load:
            units = 1000
            rev_motor = 1
    limit:
      parameter:
        v_pos = 10000.0
        v_neg = 10000.0
        a1_pos = 50000.0
        a2_pos = 50000.0
        a1_neg = 50000.0
        a2_neg = 50000.0
        t_jolt = 0.0
        t_in_pos = 0.0
        pos_sw_end = 8388607
        neg_sw_end = -8388608
        ds_warning = 500.0
        ds_stop = 1000.0
        a_stop = 1.0E+30
        dv_stop = 0.0
        dv_stop_mode = ncOFF
    controller:
      mode = ncPOSITION
      position:
        kv = 567.0
        tn = 0.0
        t_predict = 0.0004
        t_total = 0.0004
        p_max = 1.0E+30
        i_max = 0.0
      speed:
        kv = 0.25
        tn = 0.0
        t_filter = 0.0
        isq_filter1:
          type = ncOFF
          a0 = 0.0
          a1 = 0.0
          b0 = 0.0
          b1 = 0.0
          b2 = 0.0
          c0_par_id = 0
          c1_par_id = 0
        isq_filter2:
          type = ncOFF
          a0 = 0.0
          a1 = 0.0
          b0 = 0.0
          b1 = 0.0
          b2 = 0.0
          c0_par_id = 0
          c1_par_id = 0
        isq_filter3:
          type = ncOFF
          a0 = 0.0
          a1 = 0.0
          b0 = 0.0
          b1 = 0.0
          b2 = 0.0
          c0_par_id = 0
          c1_par_id = 0
      uf:
        type = ncLINEAR + ncCORRECTION
        auto_config = ncMOTOR_PAR
        u0 = 0.0
        un = 0.0
        fn = 50.0
        k_f_slip = 0.0
      ff:
        mode = ncSTANDARD
        torque_load = 0.0
        torque_pos = 0.0
        torque_neg = 0.0
        kv_torque = 0.0
        inertia = 0.0
        t_filter_a = 0.0
      fb:
        mode = ncSTANDARD
        speed_mix_ratio = 0.0
        speed_kv = 0.0
      model:
        mass1:
          inertia = 0.0
          viscous_friction = 0.0
        mass2:
          inertia = 0.0
          viscous_friction = 0.0
          stiffness = 0.0
          damping = 0.0
    move:
      stop:
        parameter[0]:
          decel_ramp = ncA_LIMIT
          controller = ncON
        parameter[1]:
          decel_ramp = ncA_LIMIT
          controller = ncON
        parameter[2]:
          decel_ramp = ncA_LIMIT
          controller = ncON
        parameter[3]:
          decel_ramp = ncA_LIMIT
          controller = ncON
        quickstop:
          decel_ramp = ncA_LIMIT
          t_jolt = 0.0
        drive_error:
          decel_ramp = ncA_LIMIT
      homing:
        parameter:
          s = 0
          v_switch = 5000.0
          v_trigger = 500.0
          a = 50000.0
          mode = ncDIRECT
          edge_sw = ncPOSITIVE
          start_dir = ncPOSITIVE
          trigg_dir = ncPOSITIVE
          ref_pulse = ncOFF
          fix_dir = ncOFF
          tr_s_block = 0.0
          torque_lim = 0.0
          ds_block = 0.0
          ds_stop = 0.0
      basis:
        parameter:
          v_pos = 5000.0
          v_neg = 5000.0
          a1_pos = 50000.0
          a2_pos = 50000.0
          a1_neg = 50000.0
          a2_neg = 50000.0
    message:
      text:
        parameter:
          format = ncBREAK
          columns = 80
          data_modul = acp10etxen
```

### Program Logical/gAxis02obj/gAxis02Basic (ANSIC) - Basic logical control

#### basic.typ - Local data types
```iecst
TYPE
	color_datapoints_typ : 	STRUCT
		color_power : INT;
		color_homing : INT;
	END_STRUCT;
	basic_command_typ : 	STRUCT  (*command structure*)
		Power : BOOL; (*switch on the controller*)
		Home : BOOL; (*reference the axis*)
		MoveAbsolute : BOOL; (*move to an defined position*)
		MoveAdditive : BOOL; (*move a defiened distance*)
		MoveVelocity : BOOL; (*start a movement with a defiened velocity*)
		Halt : BOOL; (*stop every active movement once*)
		Stop : BOOL; (*stop every active movement as long as set*)
		MoveJogPos : BOOL; (*move in positive direction as long as is set*)
		MoveJogNeg : BOOL; (*move in negative direction as long as is set*)
		ErrorAcknowledge : BOOL; (*reset active errors*)
	END_STRUCT;
	basic_parameter_typ : 	STRUCT  (*parameter structure*)
		Position : REAL; (*target-position for MoveAbsolute-Command*)
		Distance : REAL; (*distance for MoveAdditive-Command*)
		Velocity : REAL; (*velocity for MoveVelocity-Command*)
		Direction : USINT; (*direction for commanded movements*)
		Acceleration : REAL; (*acceleration for commanded movements*)
		Deceleration : REAL; (*deceleration for commanded movements*)
		HomePosition : REAL; (*target-position for referencing the axis*)
		HomeMode : USINT; (*homing mode*)
		JogVelocity : REAL; (*velocity for jogging movement*)
	END_STRUCT;
	basic_status_typ : 	STRUCT  (*status structure*)
		ErrorID : UINT; (*ErrorID of any occured error*)
		ErrorText : ARRAY[0..3]OF STRING[79]; (*Error Text*)
		ActPosition : REAL; (*actual position of the axis*)
		ActVelocity : REAL; (*actual velocity of the axis*)
		DriveStatus : MC_DRIVESTATUS_TYP; (*actual status of the axis*)
	END_STRUCT;
	basic_axisState_typ : 	STRUCT  (*axis state structure*)
		Disabled : BOOL; (*if set, axis is in state Disabled*)
		StandStill : BOOL; (*if set, axis is in state StandsStill*)
		Homing : BOOL; (*if set, axis is in state Homing*)
		Stopping : BOOL; (*if set, axis is in state Stopping*)
		DiscreteMotion : BOOL; (*if set, axis is in state DiscreteMotion*)
		ContinuousMotion : BOOL; (*if set, axis is in state ContinuousMotion*)
		SynchronizedMotion : BOOL; (*if set, axis is in state SynchronizedMotion*)
		ErrorStop : BOOL; (*if set, axis is in state ErrorStop*)
	END_STRUCT;
	basic_typ : 	STRUCT  (*control structure*)
		Command : basic_command_typ; (*command structure*)
		Parameter : basic_parameter_typ; (*parameter structure*)
		Status : basic_status_typ; (*status structure*)
		AxisState : basic_axisState_typ; (*axis state structure*)
	END_STRUCT;
END_TYPE
```

#### basic.var - Local variables
```iecst
VAR
	BasicControl : basic_typ; (*control structure*)
	Axis1Obj : UDINT; (*axis reference*)
	AxisStep : USINT; (*current step in the step sequence*)
	MC_Power_0 : MC_Power; (*Function Block*)
	MC_Home_0 : MC_Home; (*Function Block*)
	MC_Stop_0 : MC_Stop; (*Function Block*)
	MC_MoveVelocity_0 : MC_MoveVelocity; (*Function Block*)
	MC_MoveAbsolute_0 : MC_MoveAbsolute; (*Function Block*)
	MC_MoveAdditive_0 : MC_MoveAdditive; (*Function Block*)
	MC_ReadAxisError_0 : MC_ReadAxisError; (*Function Block*)
	MC_Reset_0 : MC_Reset; (*Function Block*)
	MC_ReadStatus_0 : MC_ReadStatus; (*Function Block*)
	MC_ReadActualPosition_0 : MC_ReadActualPosition; (*Function Block*)
	MC_ReadActualVelocity_0 : MC_ReadActualVelocity; (*Function Block*)
	MC_BR_ReadDriveStatus_0 : MC_BR_ReadDriveStatus; (*Function Block*)
	MC_Halt_0 : MC_Halt; (*Function Block*)
END_VAR
```

#### Init.cpp
```cpp
#ifdef _DEFAULT_INCLUDES
	#include <AsDefault.h>
#endif
#include <string.h>

#define STATE_WAIT              0

void _INIT ProgramInit(void)
{
	/* get axis object */
	Axis1Obj = (UDINT)&gAxis02;

	AxisStep = STATE_WAIT;  /* start step */

	//BasicControl.Parameter.Velocity              = 1000;  /*velocity for movement*/
	//BasicControl.Parameter.Acceleration          = 5000;  /*acceleration for movement*/
	//BasicControl.Parameter.Deceleration          = 5000;  /*deceleration for movement*/
	//BasicControl.Parameter.JogVelocity           = 400;   /*velocity for jogging */
}
```

#### Cyclic.cpp
```cpp
#ifdef _DEFAULT_INCLUDES
	#include <AsDefault.h>
#endif
#include <string.h>

/* defines of the state-constants */
#define STATE_WAIT              0
#define STATE_POWER_ON          1
#define STATE_HOME              2

#define STATE_READY             10
#define STATE_HALT              11
#define STATE_STOP              12
#define STATE_JOG_POSITIVE      13
#define STATE_JOG_NEGATIVE      14
#define STATE_MOVE_ABSOLUTE     15
#define STATE_MOVE_ADDITIVE     16
#define STATE_MOVE_VELOCITY     17

#define STATE_ERROR_AXIS        100
#define STATE_ERROR             101
#define STATE_ERROR_RESET       102

#define TWO_TICKS_JITTER 77

unsigned long bur_heap_size = 0xFFFF;

void _CYCLIC ProgramCyclic(void)
{
	/***************************************************************
        Control Sequence
	***************************************************************/

	/* status information is read before the step sequencer to attain a shorter reaction time */
	/************************ MC_READSTATUS *************************/
	MC_ReadStatus_0.Enable = !MC_ReadStatus_0.Error;
	MC_ReadStatus_0.Axis = Axis1Obj;
	MC_ReadStatus(&MC_ReadStatus_0);
	BasicControl.AxisState.Disabled             = MC_ReadStatus_0.Disabled;
	BasicControl.AxisState.StandStill           = MC_ReadStatus_0.StandStill;
	BasicControl.AxisState.Stopping             = MC_ReadStatus_0.Stopping;
	BasicControl.AxisState.Homing               = MC_ReadStatus_0.Homing;
	BasicControl.AxisState.DiscreteMotion       = MC_ReadStatus_0.DiscreteMotion;
	BasicControl.AxisState.ContinuousMotion     = MC_ReadStatus_0.ContinuousMotion;
	BasicControl.AxisState.SynchronizedMotion   = MC_ReadStatus_0.SynchronizedMotion;
	BasicControl.AxisState.ErrorStop            = MC_ReadStatus_0.Errorstop;

	/********************MC_BR_READDRIVESTATUS***********************/
	MC_BR_ReadDriveStatus_0.Enable = !MC_BR_ReadDriveStatus_0.Error;
	MC_BR_ReadDriveStatus_0.Axis = Axis1Obj;
	MC_BR_ReadDriveStatus_0.AdrDriveStatus = (UDINT)&(BasicControl.Status.DriveStatus);
	MC_BR_ReadDriveStatus(&MC_BR_ReadDriveStatus_0);

	/******************** MC_READACTUALPOSITION *********************/
	MC_ReadActualPosition_0.Enable = (!MC_ReadActualPosition_0.Error);
	MC_ReadActualPosition_0.Axis = Axis1Obj;
	MC_ReadActualPosition(&MC_ReadActualPosition_0);
	if(MC_ReadActualPosition_0.Valid == 1)
	{
		BasicControl.Status.ActPosition = MC_ReadActualPosition_0.Position;
	}

	/******************** MC_READACTUALVELOCITY *********************/
	MC_ReadActualVelocity_0.Enable = (!MC_ReadActualVelocity_0.Error);
	MC_ReadActualVelocity_0.Axis = Axis1Obj;
	MC_ReadActualVelocity(&MC_ReadActualVelocity_0);
	if(MC_ReadActualVelocity_0.Valid == 1)
	{
		BasicControl.Status.ActVelocity = MC_ReadActualVelocity_0.Velocity;
	}

	/************************ MC_READAXISERROR **********************/
	MC_ReadAxisError_0.Enable = !MC_ReadAxisError_0.Error;
	MC_ReadAxisError_0.Axis = Axis1Obj;
	MC_ReadAxisError_0.DataAddress = (UDINT)&(BasicControl.Status.ErrorText);
	MC_ReadAxisError_0.DataLength = sizeof(BasicControl.Status.ErrorText);
	strcpy(MC_ReadAxisError_0.DataObjectName,"acp10etxen");
	MC_ReadAxisError(&MC_ReadAxisError_0);

	/**************** CHECK FOR GENERAL AXIS ERROR ******************/
	if ((MC_ReadAxisError_0.AxisErrorID != 0) && (MC_ReadAxisError_0.Valid == 1))
	{
		AxisStep = STATE_ERROR_AXIS;
	}
		/***************** CHECK IF POWER SHOULD BE OFF *******************/
	else if ((BasicControl.Command.Power == 0) && (MC_ReadAxisError_0.Valid == 1))
	{
		if ((MC_ReadStatus_0.Errorstop == 1) && (MC_ReadStatus_0.Valid == 1))
		{
			AxisStep = STATE_ERROR_RESET;
		}
		else
		{
			AxisStep = STATE_WAIT;
		}
	}

	/* central monitoring of stop command attains a shorter reaction time in case of emergency stop */
	/******************CHECK for STOP COMMAND************************/
	if (BasicControl.Command.Stop == 1)
	{
		if ((AxisStep >= STATE_HOME) && (AxisStep <= STATE_ERROR))
		{
			/* reset all FB execute inputs we use */
			MC_Home_0.Execute = 0;
			MC_Stop_0.Execute = 0;
			MC_MoveAbsolute_0.Execute = 0;
			MC_MoveAdditive_0.Execute = 0;
			MC_MoveVelocity_0.Execute = 0;
			MC_Halt_0.Execute = 0;
			MC_ReadAxisError_0.Acknowledge = 0;
			MC_Reset_0.Execute = 0;

			/* reset user commands */
			BasicControl.Command.Halt = 0;
			BasicControl.Command.Home = 0;
			BasicControl.Command.MoveJogPos = 0;
			BasicControl.Command.MoveJogNeg = 0;
			BasicControl.Command.MoveVelocity = 0;
			BasicControl.Command.MoveAbsolute = 0;
			BasicControl.Command.MoveAdditive = 0;
			AxisStep = STATE_STOP;
		}
	}

	switch(AxisStep)
	{
		/******************** WAIT *************************/
		case STATE_WAIT:  /* STATE: Wait */
			if (BasicControl.Command.Power == 1)
			{
				AxisStep = STATE_POWER_ON;
			}
			else
			{
				MC_Power_0.Enable = 0;
			}

			/* reset all FB execute inputs we use */
			MC_Home_0.Execute = 0;
			MC_Stop_0.Execute = 0;
			MC_MoveAbsolute_0.Execute = 0;
			MC_MoveAdditive_0.Execute = 0;
			MC_MoveVelocity_0.Execute = 0;
			MC_Halt_0.Execute = 0;
			MC_ReadAxisError_0.Acknowledge = 0;
			MC_Reset_0.Execute = 0;

			/* reset user commands */
			BasicControl.Command.Halt = 0;
			BasicControl.Command.Home = 0;
			BasicControl.Command.MoveJogPos = 0;
			BasicControl.Command.MoveJogNeg = 0;
			BasicControl.Command.MoveVelocity = 0;
			BasicControl.Command.MoveAbsolute = 0;
			BasicControl.Command.MoveAdditive = 0;

			BasicControl.Status.ErrorID = 0;
			break;

		/******************** POWER ON **********************/
		case STATE_POWER_ON:  /* STATE: Power on */
			MC_Power_0.Enable = 1;
			if (MC_Power_0.Status == 1)
			{
				AxisStep = STATE_READY;
			}
			/* if a power error occured go to error state */
			if (MC_Power_0.Error == 1)
			{
				BasicControl.Status.ErrorID = MC_Power_0.ErrorID;
				AxisStep = STATE_ERROR;
			}
			break;

		/******************** READY **********************/
		case STATE_READY:  /* STATE: Waiting for commands */
			if (BasicControl.Command.Home == 1)
			{
				BasicControl.Command.Home = 0;
				AxisStep = STATE_HOME;
			}
			else if (BasicControl.Command.Stop == 1)
			{
				AxisStep = STATE_STOP;
			}
			else if (BasicControl.Command.MoveJogPos == 1)
			{
				AxisStep = STATE_JOG_POSITIVE;
			}
			else if (BasicControl.Command.MoveJogNeg == 1)
			{
				AxisStep = STATE_JOG_NEGATIVE;
			}
			else if (BasicControl.Command.MoveAbsolute == 1)
			{
				BasicControl.Command.MoveAbsolute = 0;
				AxisStep = STATE_MOVE_ABSOLUTE;
			}
			else if (BasicControl.Command.MoveAdditive == 1)
			{
				BasicControl.Command.MoveAdditive = 0;
				AxisStep = STATE_MOVE_ADDITIVE;
			}
			else if (BasicControl.Command.MoveVelocity == 1)
			{
				BasicControl.Command.MoveVelocity = 0;
				AxisStep = STATE_MOVE_VELOCITY;
			}
			else if (BasicControl.Command.Halt == 1)
			{
				BasicControl.Command.Halt = 0;
				AxisStep = STATE_HALT;
			}
			break;

		/******************** HOME **********************/
		case STATE_HOME:  /* STATE: start homing process */
			MC_Home_0.Position = BasicControl.Parameter.HomePosition;
			MC_Home_0.HomingMode = BasicControl.Parameter.HomeMode;
			MC_Home_0.Execute = 1;
			if (MC_Home_0.Done == 1)
			{
				MC_Home_0.Execute = 0;
				AxisStep = STATE_READY;
			}
			/* if a homing error occured go to error state */
			if (MC_Home_0.Error == 1)
			{
				MC_Home_0.Execute = 0;
				BasicControl.Status.ErrorID = MC_Home_0.ErrorID;
				AxisStep = STATE_ERROR;
			}
			break;

		/************************HALT MOVEMENT**************************/
		case STATE_HALT:  /* STATE: Stop the active movement */
			MC_Halt_0.Deceleration = BasicControl.Parameter.Deceleration;
			MC_Halt_0.Execute = 1;
			if (MC_Halt_0.Done == 1)
			{
				MC_Halt_0.Execute = 0;
				AxisStep = STATE_READY;
			}
			/*check if error occured */
			if (MC_Halt_0.Error == 1)
			{
				MC_Halt_0.Execute = 0;
				BasicControl.Status.ErrorID = MC_Halt_0.ErrorID;
				AxisStep = STATE_ERROR;
			}
			break;

		/*********************** STOP MOVEMENT *************************/
		case STATE_STOP: /* STATE: Stop movement as long as command is set */
			MC_Stop_0.Deceleration = BasicControl.Parameter.Deceleration;
			MC_Stop_0.Execute = 1;
			/* if axis is stopped go to ready state */
			if ((MC_Stop_0.Done == 1) && (BasicControl.Command.Stop == 0))
			{
				MC_Stop_0.Execute = 0;
				AxisStep = STATE_READY;
			}
			/* check if error occured */
			if (MC_Stop_0.Error == 1)
			{
				BasicControl.Status.ErrorID = MC_Stop_0.ErrorID;
				MC_Stop_0.Execute = 0;
				AxisStep = STATE_ERROR;
			}
			break;

		/******************** START JOG MOVEMENT POSITVE **********************/
		case STATE_JOG_POSITIVE:  /* STATE: Start jog movement in positive direction */
			MC_MoveVelocity_0.Velocity      = BasicControl.Parameter.JogVelocity;
			MC_MoveVelocity_0.Acceleration  = BasicControl.Parameter.Acceleration;
			MC_MoveVelocity_0.Deceleration  = BasicControl.Parameter.Deceleration;
			MC_MoveVelocity_0.Direction     = mcPOSITIVE_DIR;
			MC_MoveVelocity_0.Execute = 1;
			/* check if jog movement should be stopped */
			if (BasicControl.Command.MoveJogPos == 0)
			{
				MC_MoveVelocity_0.Execute = 0;
				AxisStep = STATE_HALT;
			}
			/* check if error occured */
			if (MC_MoveVelocity_0.Error == 1)
			{
				BasicControl.Status.ErrorID = MC_MoveVelocity_0.ErrorID;
				MC_MoveVelocity_0.Execute = 0;
				AxisStep = STATE_ERROR;
			}
			break;

		/******************** START JOG MOVEMENT NEGATIVE **********************/
		case STATE_JOG_NEGATIVE:  /* STATE: Start jog movement in negative direction */
			MC_MoveVelocity_0.Velocity      = BasicControl.Parameter.JogVelocity;
			MC_MoveVelocity_0.Acceleration  = BasicControl.Parameter.Acceleration;
			MC_MoveVelocity_0.Deceleration  = BasicControl.Parameter.Deceleration;
			MC_MoveVelocity_0.Direction     = mcNEGATIVE_DIR;
			MC_MoveVelocity_0.Execute = 1;
			/* check if jog movement should be stopped */
			if (BasicControl.Command.MoveJogNeg == 0)
			{
				MC_MoveVelocity_0.Execute = 0;
				AxisStep = STATE_HALT;
			}
			/* check if error occured */
			if (MC_MoveVelocity_0.Error == 1)
			{
				BasicControl.Status.ErrorID = MC_MoveVelocity_0.ErrorID;
				MC_MoveVelocity_0.Execute = 0;
				AxisStep = STATE_ERROR;
			}
			break;

		/******************** START ABSOLUTE MOVEMENT **********************/
		case STATE_MOVE_ABSOLUTE:  /* STATE: Start absolute movement */
			MC_MoveAbsolute_0.Position      = BasicControl.Parameter.Position;
			MC_MoveAbsolute_0.Velocity      = BasicControl.Parameter.Velocity;
			MC_MoveAbsolute_0.Acceleration  = BasicControl.Parameter.Acceleration;
			MC_MoveAbsolute_0.Deceleration  = BasicControl.Parameter.Deceleration;
			MC_MoveAbsolute_0.Direction     = BasicControl.Parameter.Direction;
			MC_MoveAbsolute_0.Execute = 1;
			/* check if commanded position is reached */
			if (BasicControl.Command.Halt == 1)
			{
				BasicControl.Command.Halt = 0;
				MC_MoveAbsolute_0.Execute = 0;
				AxisStep = STATE_HALT;
			}
			else if (MC_MoveAbsolute_0.Done == 1)
			{
				MC_MoveAbsolute_0.Execute = 0;
				AxisStep = STATE_READY;
			}
			/* check if error occured */
			if (MC_MoveAbsolute_0.Error == 1)
			{
				BasicControl.Status.ErrorID = MC_MoveAbsolute_0.ErrorID;
				MC_MoveAbsolute_0.Execute = 0;
				AxisStep = STATE_ERROR;
			}
			break;

		/******************** START ADDITIVE MOVEMENT **********************/
		case STATE_MOVE_ADDITIVE:  /* STATE: Start additive movement */
			MC_MoveAdditive_0.Distance      = BasicControl.Parameter.Distance;
			MC_MoveAdditive_0.Velocity      = BasicControl.Parameter.Velocity;
			MC_MoveAdditive_0.Acceleration  = BasicControl.Parameter.Acceleration;
			MC_MoveAdditive_0.Deceleration  = BasicControl.Parameter.Deceleration;
			MC_MoveAdditive_0.Execute = 1;
			/* check if commanded distance is reached */
			if (BasicControl.Command.Halt == 1)
			{
				BasicControl.Command.Halt = 0;
				MC_MoveAdditive_0.Execute = 0;
				AxisStep = STATE_HALT;
			}
			else if (MC_MoveAdditive_0.Done == 1)
			{
				MC_MoveAdditive_0.Execute = 0;
				AxisStep = STATE_READY;
			}
			/* check if error occured */
			if (MC_MoveAdditive_0.Error == 1)
			{
				BasicControl.Status.ErrorID = MC_MoveAdditive_0.ErrorID;
				MC_MoveAdditive_0.Execute = 0;
				AxisStep = STATE_ERROR;
			}
			break;

		/******************** START VELOCITY MOVEMENT **********************/
		case STATE_MOVE_VELOCITY:  /* STATE: Start velocity movement */
			MC_MoveVelocity_0.Velocity      = BasicControl.Parameter.Velocity;
			MC_MoveVelocity_0.Acceleration  = BasicControl.Parameter.Acceleration;
			MC_MoveVelocity_0.Deceleration  = BasicControl.Parameter.Deceleration;
			MC_MoveVelocity_0.Direction     = BasicControl.Parameter.Direction;
			MC_MoveVelocity_0.Execute = 1;
			/* check if commanded velocity is reached */
			if (BasicControl.Command.Halt == 1)
			{
				BasicControl.Command.Halt = 0;
				MC_MoveVelocity_0.Execute = 0;
				AxisStep = STATE_HALT;
			}
			else if (MC_MoveVelocity_0.InVelocity == 1)
			{
				MC_MoveVelocity_0.Execute = 0;
				AxisStep = STATE_READY;
			}
			/* check if error occured */
			if (MC_MoveVelocity_0.Error == 1)
			{
				BasicControl.Status.ErrorID = MC_MoveVelocity_0.ErrorID;
				MC_MoveVelocity_0.Execute = 0;
				AxisStep = STATE_ERROR;
			}
			break;

		/******************** FB-ERROR OCCURED *************************/
		case STATE_ERROR:  /* STATE: Error */
			/* check if FB indicates an axis error */
			if (MC_ReadAxisError_0.AxisErrorCount != 0)
			{
				AxisStep = STATE_ERROR_AXIS;
			}
			else
			{
				if (BasicControl.Command.ErrorAcknowledge == 1)
				{
					BasicControl.Command.ErrorAcknowledge = 0;
					BasicControl.Status.ErrorID = 0;
					/* reset axis if it is in axis state ErrorStop */
					if ((MC_ReadStatus_0.Errorstop == 1) && (MC_ReadStatus_0.Valid == 1))
					{
						AxisStep = STATE_ERROR_RESET;
					}
					else
					{
						AxisStep = STATE_WAIT;
					}
				}
			}
			break;

		/******************** AXIS-ERROR OCCURED *************************/
		case STATE_ERROR_AXIS:  /* STATE: Axis Error */
			if (MC_ReadAxisError_0.Valid == 1)
			{
				if (MC_ReadAxisError_0.AxisErrorID != 0)
				{
					BasicControl.Status.ErrorID = MC_ReadAxisError_0.AxisErrorID;
				}
				MC_ReadAxisError_0.Acknowledge = 0;
				if (BasicControl.Command.ErrorAcknowledge == 1)
				{
					BasicControl.Command.ErrorAcknowledge = 0;
					/* acknowledge axis error */
					if (MC_ReadAxisError_0.AxisErrorID != 0)
					{
						MC_ReadAxisError_0.Acknowledge = 1;
					}
				}
				if (MC_ReadAxisError_0.AxisErrorCount == 0)
				{
					BasicControl.Status.ErrorID = 0;
					/* reset axis if it is in axis state ErrorStop */
					if ((MC_ReadStatus_0.Errorstop == 1) && (MC_ReadStatus_0.Valid == 1))
					{
						AxisStep = STATE_ERROR_RESET;
					}
					else
					{
						AxisStep = STATE_WAIT;
					}
				}
			}
			break;

		/******************** RESET DONE *************************/
		case STATE_ERROR_RESET:  /* STATE: Wait for reset done */
			MC_Reset_0.Execute = 1;
			/* reset MC_Power.Enable if this FB is in Error*/
			if(MC_Power_0.Error == 1)
			{
				MC_Power_0.Enable = 0;
			}
			if(MC_Reset_0.Done == 1)
			{
				MC_Reset_0.Execute = 0;
				AxisStep = STATE_WAIT;
			}
			else if (MC_Reset_0.Error == 1)
			{
				MC_Reset_0.Execute = 0;
				AxisStep = STATE_ERROR;
			}
			break;

		/******************** SEQUENCE END *************************/
	}

/***************************************************************
        Function Block Calls
***************************************************************/

/************************** MC_POWER ****************************/
	MC_Power_0.Axis = Axis1Obj;  /* pointer to axis */
	MC_Power(&MC_Power_0);

	/************************** MC_HOME *****************************/
	MC_Home_0.Axis = Axis1Obj;
	MC_Home(&MC_Home_0);

	/********************** MC_MOVEABSOLUTE *************************/
	MC_MoveAbsolute_0.Axis = Axis1Obj;
	MC_MoveAbsolute(&MC_MoveAbsolute_0);

	/********************** MC_MOVEADDITIVE *************************/
	MC_MoveAdditive_0.Axis = Axis1Obj;
	MC_MoveAdditive(&MC_MoveAdditive_0);

	/********************** MC_MOVEVELOCITY *************************/
	MC_MoveVelocity_0.Axis = Axis1Obj;
	MC_MoveVelocity(&MC_MoveVelocity_0);

	/************************** MC_STOP *****************************/
	MC_Stop_0.Axis = Axis1Obj;
	MC_Stop(&MC_Stop_0);

	/**************************MC_HALT*******************************/
	MC_Halt_0.Axis = Axis1Obj;
	MC_Halt(&MC_Halt_0);

	/************************** MC_RESET ****************************/
	MC_Reset_0.Axis = Axis1Obj;
	MC_Reset(&MC_Reset_0);

	//io mapping with FieldMotor
	BasicControl.Command.Power = g_FieldMotor.IO.Power;
	BasicControl.Command.Home = g_FieldMotor.IO.Home;

	BasicControl.Command.ErrorAcknowledge = g_FieldMotor.IO.ErrorAcknowledge;
	BasicControl.Command.MoveJogNeg = g_FieldMotor.IO.MoveJogNeg;
	BasicControl.Command.MoveJogPos = g_FieldMotor.IO.MoveJogPos;
	BasicControl.Command.Stop = g_FieldMotor.IO.Stop;
	BasicControl.Command.MoveAbsolute = g_FieldMotor.IO.MoveAbsolute;

	BasicControl.Parameter.Acceleration = g_FieldMotor.IO.Acceleration;
	BasicControl.Parameter.Deceleration = g_FieldMotor.IO.Deceleration;
	BasicControl.Parameter.JogVelocity = g_FieldMotor.IO.JogVelocity;
	BasicControl.Parameter.Position = g_FieldMotor.IO.Position;
	BasicControl.Parameter.Velocity = g_FieldMotor.IO.Velocity;

	g_FieldMotor.STS.ActPosition = BasicControl.Status.ActPosition;
	if(BasicControl.Status.ActVelocity == 0 || BasicControl.Status.ActVelocity < -TWO_TICKS_JITTER || BasicControl.Status.ActVelocity > TWO_TICKS_JITTER)
	{
		g_FieldMotor.STS.ActVelocity = BasicControl.Status.ActVelocity;
	}
	g_FieldMotor.ALM.MotorError = (BasicControl.Status.ErrorID != 0);
	g_FieldMotor.ALM.ErrorID = BasicControl.Status.ErrorID;
	g_FieldMotor.STS.PowerOn = BasicControl.Command.Power;
	g_FieldMotor.STS.StandStill = BasicControl.AxisState.StandStill;

	for (int i = 0; i < 4; i++)
	{
		strncpy(
			g_FieldMotor.ALM.ErrorText[i],
			BasicControl.Status.ErrorText[i],
			sizeof(g_FieldMotor.ALM.ErrorText[i]) - 1
			);

		g_FieldMotor.ALM.ErrorText[i][sizeof(g_FieldMotor.ALM.ErrorText[i]) - 1] = '\0';
	}
}
```

### Program Logical/gAxis02obj/gAxix02Gear (ANSIC)

#### gear.c - cyclic code
```c
/*******************************************************************
 * COPYRIGHT -- Bernecker + Rainer
 ********************************************************************
 * PROGRAM: Gear
 * File: gear.c
 * Author: Bernecker + Rainer
 * Created: December 01, 2009
 ********************************************************************
 * Implementation of Program Gear
 ********************************************************************/

#ifdef _DEFAULT_INCLUDES
 #include <AsDefault.h>
#endif
#include <string.h>

/* defines for the state-variables */
#define STATE_WAIT              0
#define STATE_POWER_ON          1
#define STATE_HOME              2

#define STATE_READY             10
#define STATE_HALT              11
#define STATE_STOP              12
#define STATE_JOG_POSITIVE      13
#define STATE_JOG_NEGATIVE      14
#define STATE_MOVE_ABSOLUTE     15
#define STATE_MOVE_ADDITIVE     16
#define STATE_MOVE_VELOCITY     17

#define STATE_GEAR_START        20
#define STATE_GEAR_STOP         21

#define STATE_ERROR_AXIS        100
#define STATE_ERROR             101
#define STATE_ERROR_RESET       102

_INIT void gear_init(void)
{

/* get axis object */
Axis1Obj = (UDINT)&gAxis01;  /*Master Axis*/
Axis2Obj = (UDINT)&gAxis02;  /*Slave Axis*/

AxisStep = STATE_WAIT;  /* start step */

GearControl.Parameter.Velocity              = 1000;  /*velocity for movement*/
GearControl.Parameter.Acceleration          = 5000;  /*acceleration for movement*/
GearControl.Parameter.Deceleration          = 5000;  /*deceleration for movement*/
GearControl.Parameter.JogVelocity           = 400;   /*velocity for jogging*/
GearControl.Parameter.RatioNumerator        = 1000;  /*ratio numerator for coupling*/
GearControl.Parameter.RatioDenominator      = 1000;  /*ratio denominator for coupling*/

}

_CYCLIC void gear_cyclic(void)
{

/***************************************************************
        Control Sequence
***************************************************************/
/* status information is read before the step sequencer to attain a shorter reaction time */
/************************ MC_READSTATUS *************************/
MC_ReadStatus_0.Enable = !MC_ReadStatus_0.Error;
MC_ReadStatus_0.Axis = Axis2Obj;
MC_ReadStatus(&MC_ReadStatus_0);
GearControl.AxisState.Disabled             = MC_ReadStatus_0.Disabled;
GearControl.AxisState.StandStill           = MC_ReadStatus_0.StandStill;
GearControl.AxisState.Stopping             = MC_ReadStatus_0.Stopping;
GearControl.AxisState.Homing               = MC_ReadStatus_0.Homing;
GearControl.AxisState.DiscreteMotion       = MC_ReadStatus_0.DiscreteMotion;
GearControl.AxisState.ContinuousMotion     = MC_ReadStatus_0.ContinuousMotion;
GearControl.AxisState.SynchronizedMotion   = MC_ReadStatus_0.SynchronizedMotion;
GearControl.AxisState.ErrorStop            = MC_ReadStatus_0.Errorstop;

/********************MC_BR_READDRIVESTATUS***********************/
MC_BR_ReadDriveStatus_0.Enable = !MC_BR_ReadDriveStatus_0.Error;
MC_BR_ReadDriveStatus_0.Axis = Axis2Obj;
MC_BR_ReadDriveStatus_0.AdrDriveStatus = (UDINT)&(GearControl.Status.DriveStatus);
MC_BR_ReadDriveStatus(&MC_BR_ReadDriveStatus_0);

/******************** MC_READACTUALPOSITION *********************/
MC_ReadActualPosition_0.Enable = (!MC_ReadActualPosition_0.Error);
MC_ReadActualPosition_0.Axis = Axis2Obj;
MC_ReadActualPosition(&MC_ReadActualPosition_0);
if(MC_ReadActualPosition_0.Valid == 1)
{
    GearControl.Status.ActPosition = MC_ReadActualPosition_0.Position;
}

/******************** MC_READACTUALVELOCITY *********************/
MC_ReadActualVelocity_0.Enable = (!MC_ReadActualVelocity_0.Error);
MC_ReadActualVelocity_0.Axis = Axis2Obj;
MC_ReadActualVelocity(&MC_ReadActualVelocity_0);
if(MC_ReadActualVelocity_0.Valid == 1)
{
    GearControl.Status.ActVelocity = MC_ReadActualVelocity_0.Velocity;
}

/************************ MC_READAXISERROR **********************/
MC_ReadAxisError_0.Enable = !MC_ReadAxisError_0.Error;
MC_ReadAxisError_0.Axis = Axis2Obj;
MC_ReadAxisError_0.DataAddress = (UDINT)&(GearControl.Status.ErrorText);
MC_ReadAxisError_0.DataLength = sizeof(GearControl.Status.ErrorText);
strcpy((void*)&MC_ReadAxisError_0.DataObjectName,"acp10etxen");
MC_ReadAxisError(&MC_ReadAxisError_0);

/**************** CHECK FOR GENERAL AXIS ERROR ******************/
    if ((MC_ReadAxisError_0.AxisErrorID != 0) && (MC_ReadAxisError_0.Valid == 1))
    {
        AxisStep = STATE_ERROR_AXIS;
    }
/***************** CHECK IF POWER SHOULD BE OFF *******************/
    else if ((GearControl.Command.Power == 0) && (MC_ReadAxisError_0.Valid == 1))
    {
        if ((MC_ReadStatus_0.Errorstop == 1) && (MC_ReadStatus_0.Valid == 1))
        {
            AxisStep = STATE_ERROR_RESET;
        }
        else
        {
            AxisStep = STATE_WAIT;
        }
    }

/* central monitoring of stop command attains a shorter reaction time in case of emergency stop */
/******************CHECK for STOP COMMAND************************/
    if (GearControl.Command.Stop == 1)
    {
        if ((AxisStep >= STATE_HOME) && (AxisStep <= STATE_ERROR))
        {
            MC_Home_0.Execute = 0;
            MC_Stop_0.Execute = 0;
            MC_MoveAbsolute_0.Execute = 0;
            MC_MoveAdditive_0.Execute = 0;
            MC_MoveVelocity_0.Execute = 0;
            MC_GearIn_0.Execute = 0;
            MC_GearOut_0.Execute = 0;
            MC_Halt_0.Execute = 0;
            MC_ReadAxisError_0.Acknowledge = 0;
            MC_Reset_0.Execute = 0;

            /* reset user commands */
            GearControl.Command.Halt = 0;
            GearControl.Command.Home = 0;
            GearControl.Command.MoveJogPos = 0;
            GearControl.Command.MoveJogNeg = 0;
            GearControl.Command.MoveVelocity = 0;
            GearControl.Command.MoveAbsolute = 0;
            GearControl.Command.MoveAdditive = 0;
            GearControl.Command.StartSlave = 0;
            GearControl.Command.DisengageSlave = 0;

            AxisStep = STATE_STOP;
        }
    }

switch(AxisStep)
{
/******************** WAIT *************************/
    case STATE_WAIT:  /* STATE: Wait */
        if (GearControl.Command.Power == 1)
        {
            AxisStep = STATE_POWER_ON;
        }
        else
        {
            MC_Power_0.Enable = 0;
        }

        /* reset all FB execute inputs we use */
        MC_Home_0.Execute = 0;
        MC_Stop_0.Execute = 0;
        MC_MoveAbsolute_0.Execute = 0;
        MC_MoveAdditive_0.Execute = 0;
        MC_MoveVelocity_0.Execute = 0;
        MC_GearIn_0.Execute = 0;
        MC_GearOut_0.Execute = 0;
        MC_Halt_0.Execute = 0;
        MC_ReadAxisError_0.Acknowledge = 0;
        MC_Reset_0.Execute = 0;

        /* reset user commands */
        GearControl.Command.Stop = 0;
		GearControl.Command.Halt = 0;
        GearControl.Command.Home = 0;
        GearControl.Command.MoveJogPos = 0;
        GearControl.Command.MoveJogNeg = 0;
        GearControl.Command.MoveVelocity = 0;
        GearControl.Command.MoveAbsolute = 0;
        GearControl.Command.MoveAdditive = 0;
        GearControl.Command.StartSlave = 0;
        GearControl.Command.DisengageSlave = 0;

        GearControl.Status.ErrorID = 0;
        break;

/******************** POWER ON **********************/
    case STATE_POWER_ON:  /* STATE: Power on */
        MC_Power_0.Enable = 1;
        if (MC_Power_0.Status == 1)
        {
            AxisStep = STATE_READY;
        }
        /* if a power error occured go to error state */
        if (MC_Power_0.Error == 1)
        {
            GearControl.Status.ErrorID = MC_Power_0.ErrorID;
            AxisStep = STATE_ERROR;
        }
        break;

/******************** READY **********************/
    case STATE_READY:  /* STATE: Waiting for commands */
        if (GearControl.Command.Home == 1)
        {
            GearControl.Command.Home = 0;
            AxisStep = STATE_HOME;
        }
        else if (GearControl.Command.Stop == 1)
        {
            AxisStep = STATE_STOP;
        }
        else if (GearControl.Command.MoveJogPos == 1)
        {
            AxisStep = STATE_JOG_POSITIVE;
        }
        else if (GearControl.Command.MoveJogNeg == 1)
        {
            AxisStep = STATE_JOG_NEGATIVE;
        }
        else if (GearControl.Command.MoveAbsolute == 1)
        {
            GearControl.Command.MoveAbsolute = 0;
            AxisStep = STATE_MOVE_ABSOLUTE;
        }
        else if (GearControl.Command.MoveAdditive == 1)
        {
            GearControl.Command.MoveAdditive = 0;
            AxisStep = STATE_MOVE_ADDITIVE;
        }
        else if (GearControl.Command.MoveVelocity == 1)
        {
            GearControl.Command.MoveVelocity = 0;
            AxisStep = STATE_MOVE_VELOCITY;
        }
        else if (GearControl.Command.StartSlave == 1)
        {
            GearControl.Command.StartSlave = 0;
            AxisStep = STATE_GEAR_START;
        }
        else if (GearControl.Command.Halt == 1)
        {
            GearControl.Command.Halt = 0;
            AxisStep = STATE_HALT;
        }
        break;

/******************** HOME **********************/
    case STATE_HOME:  /* STATE: start homing process */
        MC_Home_0.Position = GearControl.Parameter.HomePosition;
        MC_Home_0.HomingMode = GearControl.Parameter.HomeMode;
        MC_Home_0.Execute = 1;
        if (MC_Home_0.Done == 1)
        {
            MC_Home_0.Execute = 0;
            AxisStep = STATE_READY;
        }
        /* if a homing error occured go to error state */
        if (MC_Home_0.Error == 1)
        {
            MC_Home_0.Execute = 0;
            GearControl.Status.ErrorID = MC_Home_0.ErrorID;
            AxisStep = STATE_ERROR;
        }
        break;

/************************HALT MOVEMENT**************************/
    case STATE_HALT:  /* STATE: Stop the active movement */
        MC_Halt_0.Deceleration = GearControl.Parameter.Deceleration;
        MC_Halt_0.Execute = 1;
        if (MC_Halt_0.Done == 1)
        {
            MC_Halt_0.Execute = 0;
            AxisStep = STATE_READY;
        }
        /*check if error occured */
        if (MC_Halt_0.Error == 1)
        {
            MC_Halt_0.Execute = 0;
            GearControl.Status.ErrorID = MC_Halt_0.ErrorID;
            AxisStep = STATE_ERROR;
        }
    break;

/*********************** STOP MOVEMENT *************************/
    case STATE_STOP:  /* STATE: Stop movement as long as command is set */
        MC_Stop_0.Deceleration = GearControl.Parameter.Deceleration;
        MC_Stop_0.Execute = 1;
        /* if axis is stopped go to ready state */
        if ((MC_Stop_0.Done == 1) && (GearControl.Command.Stop == 0))
        {
            MC_Stop_0.Execute = 0;
            AxisStep = STATE_READY;
        }
        /* check if error occured */
        if (MC_Stop_0.Error == 1)
        {
            GearControl.Status.ErrorID = MC_Stop_0.ErrorID;
            MC_Stop_0.Execute = 0;
            AxisStep = STATE_ERROR;
        }
        break;

/******************** START JOG MOVEMENT POSITVE **********************/
    case STATE_JOG_POSITIVE:  /* STATE: Start jog movement in positive direction */
        MC_MoveVelocity_0.Velocity      = GearControl.Parameter.JogVelocity;
        MC_MoveVelocity_0.Acceleration  = GearControl.Parameter.Acceleration;
        MC_MoveVelocity_0.Deceleration  = GearControl.Parameter.Deceleration;
        MC_MoveVelocity_0.Direction     = mcPOSITIVE_DIR;
        MC_MoveVelocity_0.Execute = 1;
        /* check if jog movement should be stopped */
        if (GearControl.Command.MoveJogPos == 0)
        {
            MC_MoveVelocity_0.Execute = 0;
            AxisStep = STATE_HALT;
        }
        /* check if error occured */
        if (MC_MoveVelocity_0.Error == 1)
        {
            GearControl.Status.ErrorID = MC_MoveVelocity_0.ErrorID;
            MC_MoveVelocity_0.Execute = 0;
            AxisStep = STATE_ERROR;
        }
        break;

/******************** START JOG MOVEMENT NEGATIVE **********************/
    case STATE_JOG_NEGATIVE:  /* STATE: Start jog movement in negative direction */
        MC_MoveVelocity_0.Velocity      = GearControl.Parameter.JogVelocity;
        MC_MoveVelocity_0.Acceleration  = GearControl.Parameter.Acceleration;
        MC_MoveVelocity_0.Deceleration  = GearControl.Parameter.Deceleration;
        MC_MoveVelocity_0.Direction     = mcNEGATIVE_DIR;
        MC_MoveVelocity_0.Execute = 1;
        /* check if jog movement should be stopped */
        if (GearControl.Command.MoveJogNeg == 0)
        {
            MC_MoveVelocity_0.Execute = 0;
            AxisStep = STATE_HALT;
        }
        /* check if error occured */
        if (MC_MoveVelocity_0.Error == 1)
        {
            GearControl.Status.ErrorID = MC_MoveVelocity_0.ErrorID;
            MC_MoveVelocity_0.Execute = 0;
            AxisStep = STATE_ERROR;
        }
        break;

/******************** START ABSOLUTE MOVEMENT **********************/
    case STATE_MOVE_ABSOLUTE:  /* STATE: Start absolute movement */
        MC_MoveAbsolute_0.Position      = GearControl.Parameter.Position;
        MC_MoveAbsolute_0.Velocity      = GearControl.Parameter.Velocity;
        MC_MoveAbsolute_0.Acceleration  = GearControl.Parameter.Acceleration;
        MC_MoveAbsolute_0.Deceleration  = GearControl.Parameter.Deceleration;
        MC_MoveAbsolute_0.Direction     = GearControl.Parameter.Direction;
        MC_MoveAbsolute_0.Execute = 1;
        /* check if commanded position is reached */
        if (GearControl.Command.Halt == 1)
        {
            GearControl.Command.Halt = 0;
            MC_MoveAbsolute_0.Execute = 0;
            AxisStep = STATE_HALT;
        }
        else if (MC_MoveAbsolute_0.Done == 1)
        {
            MC_MoveAbsolute_0.Execute = 0;
             AxisStep = STATE_READY;
        }
        /* check if error occured */
        if (MC_MoveAbsolute_0.Error == 1)
        {
            GearControl.Status.ErrorID = MC_MoveAbsolute_0.ErrorID;
            MC_MoveAbsolute_0.Execute = 0;
            AxisStep = STATE_ERROR;
        }
        break;

/******************** START ADDITIVE MOVEMENT **********************/
    case STATE_MOVE_ADDITIVE:  /* STATE: Start additive movement */
        MC_MoveAdditive_0.Distance      = GearControl.Parameter.Distance;
        MC_MoveAdditive_0.Velocity      = GearControl.Parameter.Velocity;
        MC_MoveAdditive_0.Acceleration  = GearControl.Parameter.Acceleration;
        MC_MoveAdditive_0.Deceleration  = GearControl.Parameter.Deceleration;
        MC_MoveAdditive_0.Execute = 1;
        /* check if commanded distance is reached */
        if (GearControl.Command.Halt == 1)
        {
            GearControl.Command.Halt = 0;
            MC_MoveAdditive_0.Execute = 0;
            AxisStep = STATE_HALT;
        }
        else if (MC_MoveAdditive_0.Done == 1)
        {
            MC_MoveAdditive_0.Execute = 0;
             AxisStep = STATE_READY;
        }
        /* check if error occured */
        if (MC_MoveAdditive_0.Error == 1)
        {
            GearControl.Status.ErrorID = MC_MoveAdditive_0.ErrorID;
            MC_MoveAdditive_0.Execute = 0;
            AxisStep = STATE_ERROR;
        }
        break;

/******************** START VELOCITY MOVEMENT **********************/
    case STATE_MOVE_VELOCITY:  /* STATE: Start velocity movement */
        MC_MoveVelocity_0.Velocity      = GearControl.Parameter.Velocity;
        MC_MoveVelocity_0.Acceleration  = GearControl.Parameter.Acceleration;
        MC_MoveVelocity_0.Deceleration  = GearControl.Parameter.Deceleration;
        MC_MoveVelocity_0.Direction     = GearControl.Parameter.Direction;
        MC_MoveVelocity_0.Execute = 1;
        /* check if commanded velocity is reached */
        if (GearControl.Command.Halt == 1)
        {
            GearControl.Command.Halt = 0;
            MC_MoveVelocity_0.Execute = 0;
            AxisStep = STATE_HALT;
        }
        else if (MC_MoveVelocity_0.InVelocity == 1)
        {
            MC_MoveVelocity_0.Execute = 0;
            AxisStep = STATE_READY;
        }
        /* check if error occured */
        if (MC_MoveVelocity_0.Error == 1)
        {
            GearControl.Status.ErrorID = MC_MoveVelocity_0.ErrorID;
            MC_MoveVelocity_0.Execute = 0;
            AxisStep = STATE_ERROR;
        }
        break;

/******************** START GEAR MOVEMENT **********************/
    case STATE_GEAR_START:  /* STATE: Start electronic gear coupling */
        MC_GearIn_0.RatioNumerator   = GearControl.Parameter.RatioNumerator;
        MC_GearIn_0.RatioDenominator = GearControl.Parameter.RatioDenominator;
        MC_GearIn_0.Acceleration     = GearControl.Parameter.Acceleration;
        MC_GearIn_0.Deceleration     = GearControl.Parameter.Deceleration;
        MC_GearIn_0.Execute = 1;
        /* wait for gear stop */
        if (GearControl.Command.Halt == 1)
        {
            GearControl.Command.Halt = 0;
            MC_GearIn_0.Execute = 0;
            AxisStep = STATE_HALT;
        }
        else if (GearControl.Command.DisengageSlave == 1)
        {
            GearControl.Command.DisengageSlave = 0;
            MC_GearIn_0.Execute = 0;
            AxisStep = STATE_GEAR_STOP;
        }
        /* check if error occured */
        if (MC_GearIn_0.Error == 1)
        {
            GearControl.Status.ErrorID = MC_GearIn_0.ErrorID;
            MC_GearIn_0.Execute = 0;
            AxisStep = STATE_ERROR;
        }
        break;

/******************** STOP GEAR MOVEMENT **********************/
    case STATE_GEAR_STOP:  /* STATE: Stop electronic gear coupling */
        MC_GearOut_0.Execute = 1;
        /* check if coupling is stopped */
        if (MC_GearOut_0.Done == 1)
        {
            MC_GearOut_0.Execute = 0;
            AxisStep = STATE_READY;
        }
        /* check if error occured */
        if (MC_GearOut_0.Error == 1)
        {
            GearControl.Status.ErrorID = MC_GearOut_0.ErrorID;
            MC_GearOut_0.Execute = 0;
            AxisStep = STATE_ERROR;
        }
        break;

/******************** FB-ERROR OCCURED *************************/
    case STATE_ERROR:  /* STATE: Error */
        /* check if FB indicates an axis error */
        if (MC_ReadAxisError_0.AxisErrorCount != 0)
        {
            AxisStep = STATE_ERROR_AXIS;
        }
        else
        {
            if (GearControl.Command.ErrorAcknowledge == 1)
            {
                GearControl.Command.ErrorAcknowledge = 0;
                GearControl.Status.ErrorID = 0;
                /* reset axis if it is in axis state ErrorStop */
                if ((MC_ReadStatus_0.Errorstop == 1) && (MC_ReadStatus_0.Valid == 1))
                {
                    AxisStep = STATE_ERROR_RESET;
                }
                else
                {
                    AxisStep = STATE_WAIT;
                }
            }
        }
        break;

/******************** AXIS-ERROR OCCURED *************************/
    case STATE_ERROR_AXIS:  /* STATE: Axis Error */
        if (MC_ReadAxisError_0.Valid == 1)
        {
            if (MC_ReadAxisError_0.AxisErrorID != 0)
            {
                GearControl.Status.ErrorID = MC_ReadAxisError_0.AxisErrorID;
            }
            MC_ReadAxisError_0.Acknowledge = 0;
            if (GearControl.Command.ErrorAcknowledge == 1)
            {
                GearControl.Command.ErrorAcknowledge = 0;
                /* acknowledge axis error */
                if (MC_ReadAxisError_0.AxisErrorID != 0)
                {
                    MC_ReadAxisError_0.Acknowledge = 1;
                }
            }
            if (MC_ReadAxisError_0.AxisErrorCount == 0)
            {
                GearControl.Status.ErrorID = 0;
                /* reset axis if it is in axis state ErrorStop */
                if ((MC_ReadStatus_0.Errorstop == 1) && (MC_ReadStatus_0.Valid == 1))
                {
                    AxisStep = STATE_ERROR_RESET;
                }
                else
                {
                    AxisStep = STATE_WAIT;
                }
            }
        }
        break;

/******************** RESET DONE *************************/
    case STATE_ERROR_RESET:  /* STATE: Wait for reset done */
        MC_Reset_0.Execute = 1;
        /* reset MC_Power.Enable if this FB is in Error*/
        if(MC_Power_0.Error == 1)
        {
            MC_Power_0.Enable = 0;
        }
        if(MC_Reset_0.Done == 1)
        {
            MC_Reset_0.Execute = 0;
            AxisStep = STATE_WAIT;
        }
        else if(MC_Reset_0.Error == 1)
        {
            MC_Reset_0.Execute = 0;
            AxisStep = STATE_ERROR;
        }
        break;
/******************** SEQUENCE END *************************/
}

/***************************************************************
        Function Block Calls
***************************************************************/

/************************** MC_POWER ****************************/
MC_Power_0.Axis = Axis2Obj; /* pointer to axis */
MC_Power(&MC_Power_0);

/************************** MC_HOME *****************************/
MC_Home_0.Axis = Axis2Obj;
MC_Home(&MC_Home_0);

/********************** MC_MOVEABSOLUTE *************************/
MC_MoveAbsolute_0.Axis = Axis2Obj;
MC_MoveAbsolute(&MC_MoveAbsolute_0);

/********************** MC_MOVEADDITIVE *************************/
MC_MoveAdditive_0.Axis = Axis2Obj;
MC_MoveAdditive(&MC_MoveAdditive_0);

/********************** MC_MOVEVELOCITY *************************/
MC_MoveVelocity_0.Axis = Axis2Obj;
MC_MoveVelocity(&MC_MoveVelocity_0);

/********************** MC_GEARIN *************************/
MC_GearIn_0.Master = Axis1Obj;
MC_GearIn_0.Slave = Axis2Obj;
MC_GearIn(&MC_GearIn_0);

/********************** MC_GEAROUT *************************/
MC_GearOut_0.Slave = Axis2Obj;
MC_GearOut(&MC_GearOut_0);

/************************** MC_STOP *****************************/
MC_Stop_0.Axis = Axis2Obj;
MC_Stop(&MC_Stop_0);

/**************************MC_HALT*******************************/
MC_Halt_0.Axis = Axis2Obj;
MC_Halt(&MC_Halt_0);

/************************** MC_RESET ****************************/
MC_Reset_0.Axis = Axis2Obj;
MC_Reset(&MC_Reset_0);

}
```

#### gear.typ - Local data types
```iecst
TYPE
	gear_command_typ : 	STRUCT  (*command structure*)
		Power : BOOL; (*switch on the controller*)
		Home : BOOL; (*reference the axis*)
		MoveAbsolute : BOOL; (*move to an defined position*)
		MoveAdditive : BOOL; (*move a defiened distance*)
		MoveVelocity : BOOL; (*start a movement with a defiened velocity*)
		Halt : BOOL; (*stop every active movement*)
		Stop : BOOL; (*stop every active movement as long as is set*)
		MoveJogPos : BOOL; (*move in positive direction as long as is set*)
		MoveJogNeg : BOOL; (*move in negative direction as long as is set*)
		StartSlave : BOOL; (*start coupling beetween master and slave*)
		DisengageSlave : BOOL; (*stop coupling between master and slave*)
		ErrorAcknowledge : BOOL; (*reset active errors*)
	END_STRUCT;
	gear_parameter_typ : 	STRUCT  (*parameter structure*)
		Position : REAL; (*target-position for MoveAbsolute-Command*)
		Distance : REAL; (*distance for MoveAdditive-Command*)
		Velocity : REAL; (*velocity for MoveVelocity-Command*)
		Direction : USINT; (*direction for commanded movements*)
		Acceleration : REAL; (*acceleration for commanded movements*)
		Deceleration : REAL; (*deceleration for commanded movements*)
		HomePosition : REAL; (*target-position for referencing the axis*)
		HomeMode : USINT; (*homing mode*)
		JogVelocity : REAL; (*velocity for jogging movement*)
		RatioNumerator : INT; (*ratio numerator for coupling*)
		RatioDenominator : UINT; (*ratio denominator for coupling*)
	END_STRUCT;
	gear_status_typ : 	STRUCT  (*status structure*)
		ErrorID : UINT; (*ErrorID of any occured error*)
		ErrorText : ARRAY[0..3] OF STRING[79]; (*Error Text*)
		ActPosition : REAL; (*actual position of the axis*)
		ActVelocity : REAL; (*actual velocity of the axis*)
		DriveStatus : MC_DRIVESTATUS_TYP; (*actual status of the axis*)
	END_STRUCT;
	gear_axisState_typ : 	STRUCT  (*axis state structure*)
		Disabled : BOOL; (*if set, axis is in state Disabled*)
		StandStill : BOOL; (*if set, axis is in state StandsStill*)
		Homing : BOOL; (*if set, axis is in state Homing*)
		Stopping : BOOL; (*if set, axis is in state Stopping*)
		DiscreteMotion : BOOL; (*if set, axis is in state DiscreteMotion*)
		ContinuousMotion : BOOL; (*if set, axis is in state ContinuousMotion*)
		SynchronizedMotion : BOOL; (*if set, axis is in state SynchronizedMotion*)
		ErrorStop : BOOL; (*if set, axis is in state ErrorStop*)
	END_STRUCT;
	gear_typ : 	STRUCT  (*control structure*)
		Command : gear_command_typ; (*command structure*)
		Parameter : gear_parameter_typ; (*parameter structure*)
		Status : gear_status_typ; (*status structure*)
		AxisState : gear_axisState_typ; (*axis state strucutre*)
	END_STRUCT;
END_TYPE
```

#### gear.var - Local variables
```iecst
VAR
	GearControl : gear_typ; (*control structure*)
	Axis1Obj : UDINT; (*axis reference*)
	Axis2Obj : UDINT; (*axis reference*)
	AxisStep : USINT; (*current step in the step sequence*)
	MC_Power_0 : MC_Power; (*Function Block*)
	MC_Home_0 : MC_Home; (*Function Block*)
	MC_Stop_0 : MC_Stop; (*Function Block*)
	MC_MoveVelocity_0 : MC_MoveVelocity; (*Function Block*)
	MC_MoveAbsolute_0 : MC_MoveAbsolute; (*Function Block*)
	MC_MoveAdditive_0 : MC_MoveAdditive; (*Function Block*)
	MC_GearIn_0 : MC_GearIn; (*Function Block*)
	MC_GearOut_0 : MC_GearOut; (*Function Block*)
	MC_ReadAxisError_0 : MC_ReadAxisError; (*Function Block*)
	MC_Reset_0 : MC_Reset; (*Function Block*)
	MC_ReadStatus_0 : MC_ReadStatus; (*Function Block*)
	MC_ReadActualPosition_0 : MC_ReadActualPosition; (*Function Block*)
	MC_ReadActualVelocity_0 : MC_ReadActualVelocity; (*Function Block*)
	MC_BR_ReadDriveStatus_0 : MC_BR_ReadDriveStatus; (*Function Block*)
	MC_Halt_0 : MC_Halt; (*Function Block*)
END_VAR
```

- Visualisation Logical/Visu (not shown)

### Program Logical/UnitTests/UnitTests/Tests_FieldMotor_C (ANSIC) - Empty template for use with helper tool

#### variables.var - Name the suite and add PVs for the program
```iecst
(********************************************************************
 * COPYRIGHT --  MyAutomation-IT
 ********************************************************************
 * Program: Tests_FieldMotor_C
 * File: variables.var
 * Author: Raivo Berends
 ********************************************************************
 * Local variables of program Tests_FieldMotor_C
 ********************************************************************)
(*Describe the test*)
VAR
	Testsuite : UtMgrTestSuite := (Name:='FieldMotor_Tests',Type:=utMgrTEST_TYPE_C);
END_VAR
(*Variables used in the tests*)
VAR
	FieldMotorFB : FB_FieldMotor;
	FieldMotorStruct : UDT_FieldMotor;
END_VAR
```

#### autoGeneratedFile.c - Auto generated code - list of all test sets in the program
```c
/*
B+R UnitTest: This is generated code.
Do not edit! Do not move!
Description: UnitTest Testprogramm infrastructure (List of TestSets).
LastUpdated: 2026-05-07 09:03:54Z
By B+R UnitTest Helper Version: 2.0.2.35
*/
#include "UnitTest.h"

UNITTEST_TESTSET_DECLARATION  testSet_FieldMotor_Disabled;
UNITTEST_TESTSET_DECLARATION  testSet_FieldMotor_Initializing;
UNITTEST_TESTSET_DECLARATION  testSet_FieldMotor_Idle;
UNITTEST_TESTSET_DECLARATION  testSet_FieldMotor_Running;
UNITTEST_TESTSET_DECLARATION  testSet_FieldMotor_Stopping;

UNITTEST_TESTSET_FIXTURES(utTestSets)
{
	new_TestSet(testSet_FieldMotor_Disabled),
	new_TestSet(testSet_FieldMotor_Initializing),
	new_TestSet(testSet_FieldMotor_Idle),
	new_TestSet(testSet_FieldMotor_Running),
	new_TestSet(testSet_FieldMotor_Stopping),
};
UNTITTEST_TESTSET_HANDLER();
```
